(* Logix 5000 project; controller PBS_Perfusion vendor 1 type 14 code 217 rev 32.14; software revision 32.03; part 19 of 27 *)
(* tags used below, declared in another part *)
   Out_Open : BOOL;   // Pulse Output to drive valve Open
   Out_Close : BOOL;   // Pulse Output to drive valve closed
   P_ValveC : BOOL;   // Unique Parameter Name for auto - discovery
   OCmd_BumpClose : BOOL;   // Operator Command to bump valve closed (avail. if Fdbk Bad)
   OCmd_BumpOpen : BOOL;   // Operator Command to bump valve open (avail. if Fdbk Bad)
   ORdy_CV : BOOL;   // 1=Ready for OSet_CV (enables data entry field)
   ORdy_BumpClose : BOOL;   // 1=Ready for OCmd_BumpClose (enables HMI button)
   ORdy_BumpOpen : BOOL;   // 1=Ready for OCmd_BumpOpen (enables HMI button)
   REAL : DINT;
(* P_ValveC, continued *)

ROUTINE Prescan   (* ladder *)
// Clear Ownership. clear "lurking" Commands
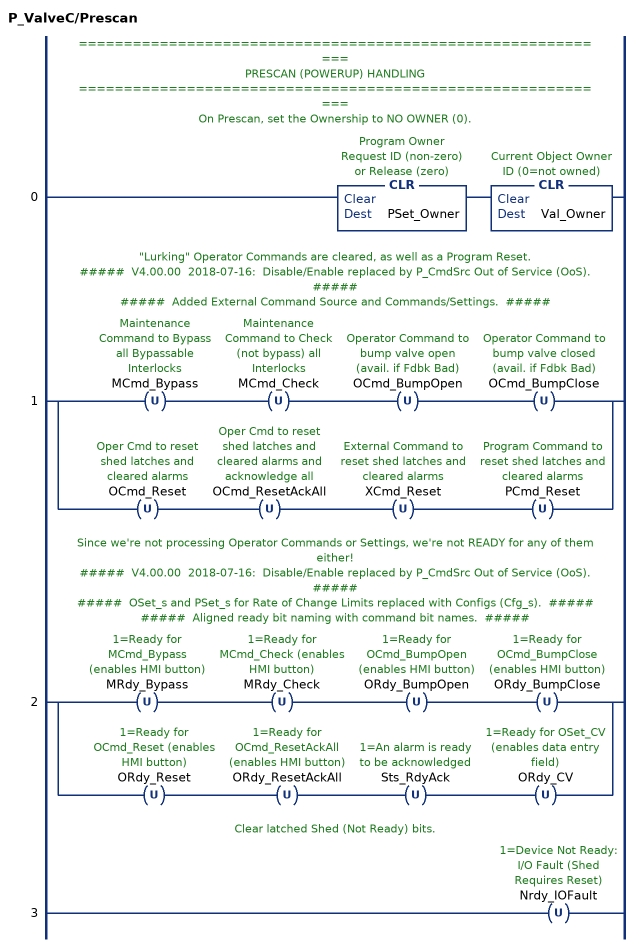
   // ============================================================
   // PRESCAN (POWERUP) HANDLING
   // ============================================================
   // On Prescan, set the Ownership to NO OWNER (0).
   0: CLR(PSet_Owner)CLR(Val_Owner);
   // "Lurking" Operator Commands are cleared, as well as a Program Reset.
   // #####  V4.00.00  2018-07-16:  Disable/Enable replaced by P_CmdSrc Out of Service (OoS).  #####
   // #####  Added External Command Source and Commands/Settings.  #####
   1: [OTU(MCmd_Bypass) OTU(MCmd_Check) OTU(OCmd_BumpOpen) OTU(OCmd_BumpClose) ,OTU(OCmd_Reset) OTU(OCmd_ResetAckAll) OTU(XCmd_Reset) OTU(PCmd_Reset) ];
   // Since we're not processing Operator Commands or Settings, we're not READY for any of them either!
   // #####  V4.00.00  2018-07-16:  Disable/Enable replaced by P_CmdSrc Out of Service (OoS).  #####
   // #####  OSet_s and PSet_s for Rate of Change Limits replaced with Configs (Cfg_s).  #####
   // #####  Aligned ready bit naming with command bit names.  #####
   2: [OTU(MRdy_Bypass) OTU(MRdy_Check) OTU(ORdy_BumpOpen) OTU(ORdy_BumpClose) ,OTU(ORdy_Reset) OTU(ORdy_ResetAckAll) OTU(Sts_RdyAck) OTU(ORdy_CV) ];
   // Clear latched Shed (Not Ready) bits.
   3: OTU(Nrdy_IOFault);
END_ROUTINE
END_ADD_ON_INSTRUCTION

ADD_ON_INSTRUCTION P_ValveSO   (* revision 4.10 .01 Release, vendor Rockwell Automation, ExecutePrescan, ExecuteEnableInFalse *)
// Solenoid Operated Valve
// Revision note:
// See Instruction Help for a summary of changes, and see 4.10 Release Notes for details.
// Help:
// Copyright © Rockwell Automation, Inc.  All Rights Reserved.
// This Instruction controls and monitors a single solenoid operated
// valve (two position: opened, closed) and provides:
// *  Support for fail open (energize to close) and fail closed (energize to open, default) valves
// *  Monitoring of limit switch feedback, display of actual valve status
// *  Detection of Failure to Open, Failure to Close
// *  Monitoring of Permissive conditions to allow energizing
// *  Monitoring of Interlock conditions to de-energize
// *  Simulation, providing feedback of a working valve while disabling outputs
// *  Monitoring of I/O communication faults
// *  Alarms for Full Stall (didn't move), Transit Stall (didn't reach target position), Interlock Trip, I/O Fault
// *  Operation in Hand, Maintenance, Override, Program and Operator Modes
// *  "Available" status for use by automation logic to know whether valve
//       can be controlled by other objects.
// Command Sources are arbitrated by a P_CmdSrc Add-On Instruction instance.
// Command Sources: Operator, External, Program, Override, Maintenance, Out of
// Service, Hand.  Alarms are provided by P_Alarm Add-On Instruction instances.
// SUMMARY OF CHANGES FROM PREVIOUS VERSION (4.10.00)
// See 4.10 Release Notes for details.
// * No changes, uprevved because P_CmdSrc 4.10.01 is used.
// SUMMARY OF CHANGES FROM PREVIOUS VERSION (4.00.02)
// See 4.10 Release Notes for details.
// * Added audible alert on commanded energize.
// * Added Horn Status, Horn Inhibit.
// * Updated to P_CmdSrc V4.10.00.
// * Added Cfg_HasMoreObj.
// SUMMARY OF CHANGES FROM PREVIOUS VERSION (4.00.01)
// See 4.00 Release Notes for details.
// * Modified handling of simultaneous open and close commands.
// SUMMARY OF CHANGES FROM PREVIOUS VERSION (4.00.00)
// See 4.00 Release Notes for details.
// * Corrected Reset Command logic.
// SUMMARY OF CHANGES FROM PREVIOUS VERSION (3.5-11)
// See 4.00 Release Notes for details.
// * Changed Inf_ items to HMI_, and added Cfg_Area for security.
// * Added notify and unack count rollup for Channel object.
// * Changed "Mode" to "Command Source" using P_CmdSrc 4.00.00.
// * Deleted Cfg_PCmdClear; all Program Commands are now self-clearing.
// * Aligned ready bit naming with command bit names.
// * All OCmds/MCmds and ORdys/MRdys are now Local Tags.
// * Added Sts_RdyAck and Sts_RdyReset for use by external objects.
// * Changed delay / time configuration items to REAL seconds.
VAR_INPUT
   Inp_OpenLS : BOOL; {visible}   // Valve Open Limit Switch 1=confirmed OPEN
   Inp_ClosedLS : BOOL; {visible}   // Valve Closed Limit Switch 1=confirmed CLOSED
   Inp_PermOK : BOOL := 1; {visible}   // 1=Permissives OK, Valve can energize
   Inp_NBPermOK : BOOL := 1; {visible}   // 1=Non-Bypassable Permissives OK, valve can energize
   Inp_IntlkOK : BOOL := 1; {visible}   // 1=Interlocks OK, valve can energize
   Inp_NBIntlkOK : BOOL := 1; {visible}   // 1=Non-Bypassable Interlocks OK, valve can energize
   Inp_IntlkAvail : BOOL;   // 1 = Interlock Availibility OK
   Inp_IOFault : BOOL;   // Input Communication Status 0=OK, 1=fail
   Inp_Sim : BOOL;   // 1=Simulate working valve; 0=Open/Close/ Monitor actual valve
   Inp_Hand : ALIAS FOR CmdSrc.Inp_Hand;
   Inp_Ovrd : ALIAS FOR CmdSrc.Inp_Ovrd;
   Inp_OvrdCmd : DINT;   // Override Mode Command: 0=None, 1=Close, 2=Open
   Inp_ExtInh : ALIAS FOR CmdSrc.Inp_ExtInh;
   Inp_HornInh : BOOL;   // 1 = Inhibit audible alert, 0 = Alllow audible alert
   Inp_Reset : BOOL;   // 1=Reset all fault conditions and latched Alarms
   Cfg_FailOpen : BOOL;   // 1=Fail Open (energize to close), 0=Fail Closed (energize to open)
   Cfg_HasOpenLS : BOOL;   // 1=Valve provides an Open Limit Switch signal
   Cfg_HasClosedLS : BOOL;   // 1=Valve provides a Closed Limit Switch signal
   Cfg_UseOpenLS : BOOL;   // 1=Valve Open LS should be used for failure checking
   Cfg_UseClosedLS : BOOL;   // 1=Valve Closed LS should be used for failure checking
   Cfg_LSFail : BOOL := 1;   // 1=both switches ON=fail, 0=both switches OFF=fail
   Cfg_HasPermObj : BOOL;   // 1=Tells HMI a P_Perm is connected to Inp_Perm
   Cfg_HasIntlkObj : BOOL;   // 1=Tells HMI a P_Intlk is connected to Inp_Intlk
   Cfg_HasStatsObj : BOOL;   // 1=Tells HMI a P_ValveStats is monitoring this valve
   Cfg_HasMoreObj : BOOL;   // 1=Tells HMI an object with more info is available
   Cfg_OCmdResets : BOOL;   // 1=New valve OCmd resets shed latches and cleared alarms, 0=OCmdReset req'd.
   Cfg_XCmdResets : BOOL;   // 1=New valve XCmd resets shed latches and cleared alarms, 0=OCmdReset req'd.
   Cfg_OvrdPermIntlk : BOOL;   // 1=Override ignores Bypassable Perm/ Intlk; 0=always use Perm/Intlk
   Cfg_ShedOnFullStall : BOOL := 1;   // 1=Stop Valve and Alarm on Full Stall; 0=Alarm only on Full Stall
   Cfg_ShedOnTransitStall : BOOL := 1;   // 1=Stop Valve and Alarm on Transit Stall; 0=Alarm only on Transit Stall
   Cfg_ShedOnIOFault : BOOL := 1;   // 1=Stop Valve and Alarm on I/O Fault; 0=Alarm only on I/O Fault
   Cfg_HasFullStallAlm : ALIAS FOR FullStall.Cfg_Exists;   // 1=Full Stall Alarm exists and will be checked
   Cfg_HasTransitStallAlm : ALIAS FOR TransitStall.Cfg_Exists;   // 1=Transit Stall Alarm exists and will be checked
   Cfg_HasIntlkTripAlm : ALIAS FOR IntlkTrip.Cfg_Exists;   // 1=Interlock Trip Alarm exists and will be checked
   Cfg_HasIOFaultAlm : ALIAS FOR IOFault.Cfg_Exists;   // 1=I/O Fault Alarm exists and will be checked
   Cfg_FullStallResetReqd : ALIAS FOR FullStall.Cfg_ResetReqd;   // 1=Reset requied to clear Full Stall Alarm
   Cfg_TransitStallResetReqd : ALIAS FOR TransitStall.Cfg_ResetReqd;   // 1=Reset required to clear Transit Stall Alarm
   Cfg_IntlkTripResetReqd : ALIAS FOR IntlkTrip.Cfg_ResetReqd;   // 1=Reset required to clear Interlock Trip Alarm
   Cfg_IOFaultResetReqd : ALIAS FOR IOFault.Cfg_ResetReqd;   // 1=Reset required to clear I/O Fault Alarm
   Cfg_FullStallAckReqd : ALIAS FOR FullStall.Cfg_AckReqd;   // 1=Acknowledge required for Full Stall Alarm
   Cfg_TransitStallAckReqd : ALIAS FOR TransitStall.Cfg_AckReqd;   // 1=Acknowledge required for Transit Stall Alarm
   Cfg_IntlkTripAckReqd : ALIAS FOR IntlkTrip.Cfg_AckReqd;   // 1=Acknowledge required for Interlock Trip Alarm
   Cfg_IOFaultAckReqd : ALIAS FOR IOFault.Cfg_AckReqd;   // 1=Acknowledge required for I/O Fault Alarm
   Cfg_FullStallSeverity : ALIAS FOR FullStall.Cfg_Severity;   // Full Stall Alarm Severity: 1..250=Low, 251..500=Medium, 501..750=High, 751..1000=Urgent
   Cfg_TransitStallSeverity : ALIAS FOR TransitStall.Cfg_Severity;   // Transit Stall Alarm Severity: 1..250=Low, 251..500=Medium, 501..750=High, 751..1000=Urgent
   Cfg_IntlkTripSeverity : ALIAS FOR IntlkTrip.Cfg_Severity;   // Interlock Trip Alarm Severity: 1..250=Low, 251..500=Medium, 501..750=High, 751..1000=Urgent
   Cfg_IOFaultSeverity : ALIAS FOR IOFault.Cfg_Severity;   // I/O Fault Alarm Severity: 1..250=Low, 251..500=Medium, 501..750=High, 751..1000=Urgent
   Cfg_SimFdbkT : REAL := 2.0;   // Delay to echo back of Open/Closed status when in Simulation (sec)
   Cfg_FullStallT : REAL := 5.0;   // After command, time with no motion before Fault (sec)
   Cfg_TransitStallT : REAL := 10.0;   // After command, time to reach position before fault (sec)
   Cfg_StartHornT : REAL;   // Time to sound audible on commanded start (sec) (0=disabled)
   PSet_Owner : DINT;   // Program Owner Request ID (non-zero) or Release (zero)
   PCmd_Open : BOOL;   // Program Command to Open Valve
   PCmd_Close : BOOL;   // Program Command to Close Valve
   PCmd_Prog : ALIAS FOR CmdSrc.PCmd_Prog;
   PCmd_Oper : ALIAS FOR CmdSrc.PCmd_Oper;
   PCmd_Lock : ALIAS FOR CmdSrc.PCmd_Lock;
   PCmd_Unlock : ALIAS FOR CmdSrc.PCmd_Unlock;
   PCmd_Normal : ALIAS FOR CmdSrc.PCmd_Normal;
   PCmd_Reset : BOOL;   // Program Command to ResetShed Latches and Cleared Alarms
   PCmd_FullStallAck : ALIAS FOR FullStall.PCmd_Ack;   // Program Command to Acknowledge Full Stall Alarm
   PCmd_FullStallSuppress : ALIAS FOR FullStall.PCmd_Suppress;   // Program Command to Suppress Full Stall Alarm
   PCmd_FullStallUnsuppress : ALIAS FOR FullStall.PCmd_Unsuppress;   // Program Command to Unsuppress Full Stall Alarm
   PCmd_FullStallUnshelve : ALIAS FOR FullStall.PCmd_Unshelve;   // Program Command to Unshelve Full Stall Alarm
   PCmd_TransitStallAck : ALIAS FOR TransitStall.PCmd_Ack;   // Program Command to Acknowledge Transit Stall Alarm
   PCmd_TransitStallSuppress : ALIAS FOR TransitStall.PCmd_Suppress;   // Program Command to Suppress Transit Stall Alarm
   PCmd_TransitStallUnsuppress : ALIAS FOR TransitStall.PCmd_Unsuppress;   // Program Command to Unsuppress Transit Stall Alarm
   PCmd_TransitStallUnshelve : ALIAS FOR TransitStall.PCmd_Unshelve;   // Program Command to Unshelve Transit Stall Alarm
   PCmd_IntlkTripAck : ALIAS FOR IntlkTrip.PCmd_Ack;   // Program Command to Acknowledge Interlock Trip Alarm
   PCmd_IntlkTripSuppress : ALIAS FOR IntlkTrip.PCmd_Suppress;   // Program Command to Suppress Interlock Trip Alarm
   PCmd_IntlkTripUnsuppress : ALIAS FOR IntlkTrip.PCmd_Unsuppress;   // Program Command to Unsuppress Interlock Trip Alarm
   PCmd_IntlkTripUnshelve : ALIAS FOR IntlkTrip.PCmd_Unshelve;   // Program Command to Unshelve Interlock Trip Alarm
   PCmd_IOFaultAck : ALIAS FOR IOFault.PCmd_Ack;   // Program Command to Acknowledge I/O Fault Alarm
   PCmd_IOFaultSuppress : ALIAS FOR IOFault.PCmd_Suppress;   // Program Command to Suppress I/O Fault Alarm
   PCmd_IOFaultUnsuppress : ALIAS FOR IOFault.PCmd_Unsuppress;   // Program Command to Unsuppress I/O Fault Alarm
   PCmd_IOFaultUnshelve : ALIAS FOR IOFault.PCmd_Unshelve;   // Program Command to Unshelve I/O Fault Alarm
   MCmd_Rel : ALIAS FOR CmdSrc.MCmd_Rel;
   OCmd_Unlock : ALIAS FOR CmdSrc.OCmd_Unlock;
   XCmd_Open : BOOL;   // External Command to Open Valve
   XCmd_Close : BOOL;   // External Command to Close Valve
   XCmd_Acq : ALIAS FOR CmdSrc.XCmd_Acq;
   XCmd_Rel : ALIAS FOR CmdSrc.XCmd_Rel;
   XCmd_Reset : BOOL;   // Ext Cmd to clear shed latches and cleared alarms
END_VAR
VAR_OUTPUT
   Out : BOOL; {access Read Only, visible}   // 1=Energize Valve Solenoid
   Out_Horn : BOOL; {access Read Only, visible}   // 1=Sound audible prior to commanded motor start
   SrcQ_IO : DINT; {access Read Only}   // Source and Quality of primary I/O (enumeration)
   SrcQ : DINT; {access Read Only}   // Source and Quality of primary Val/Sts (enumeration)
   Val_Cmd : DINT; {access Read Only}   // Device Command 0=None, 1=Close, 2=Open
   Val_Fdbk : DINT; {access Read Only}   // Device Feedback 0=Moving, 1=Closed, 2=Opened, 3=Limit Switch Failure
   Val_Sts : DINT; {access Read Only}   // Device Confirmed Sts 0=? 1=Closed 2=Open 5=Closing, 6=Opening
   Val_Fault : DINT; {access Read Only}   // Device Fault Status 0=None, 16=Transit Stall, 17 = Full Stall, 32=I/O Fault, 34=Config Error
   Val_NotifyAll : DINT; {access Read Only}   // Highest Alarm prio and ack status this object + channel (enum)
   Val_UnackAlmC : DINT; {access Read Only}   // Count of Unacknowledged Alarms
   Val_Owner : DINT; {access Read Only}   // Current Object Owner ID (0=not owned)
   Sts_Closed : BOOL; {access Read Only, visible}   // 1=Valve requested to Close and is confirmed Closed
   Sts_Opening : BOOL; {access Read Only, visible}   // 1=Valve requested to open and awaiting open feedback
   Sts_Opened : BOOL; {access Read Only, visible}   // 1=Valve requested to open and is confirmed Opened
   Sts_Closing : BOOL; {access Read Only, visible}   // 1=Valve requested to Close and awaiting Closed feedback
   Sts_Horn : BOOL; {access Read Only}   // 1=Valve Horn Active
   Sts_Available : BOOL; {access Read Only}   // 1=Valve available for control by automation (Prog)
   Sts_Bypass : BOOL; {access Read Only}   // 1=Bypassable Interlocks and Permissives are Bypassed
   Sts_BypActive : BOOL; {access Read Only}   // 1=Bypassing Active (Bypassed or Maintenance)
   Sts_LSFail : BOOL; {access Read Only}   // 1=Limit Switch Overlap Failure
   Sts_NotRdy : BOOL; {access Read Only}   // 1=Device Not Ready, see detail bits for reason
   Nrdy_CfgErr : BOOL; {access Read Only}   // 1=Device Not Ready: Configuration Error
   Nrdy_Fail : BOOL; {access Read Only}   // 1=Device Not Ready: Device Failure (Shed Requires Reset)
   Nrdy_Intlk : BOOL; {access Read Only}   // 1=Device Not Ready: Interlock Not OK
   Nrdy_IOFault : BOOL; {access Read Only}   // 1=Device Not Ready: I/O Fault (Shed Requires Reset)
   Nrdy_OoS : BOOL; {access Read Only}   // 1=Device Not Ready: Device is Out of Service
   Nrdy_Perm : BOOL; {access Read Only}   // 1=Device Not Ready: Permissive Not OK
   Sts_MaintByp : BOOL; {access Read Only}   // 1=A Maintenance Bypass is Active, display icon
   Sts_AlmInh : BOOL; {access Read Only}   // 1=An Alarm is Shelved, Disabled or Suppressed, display icon
   Sts_Err : BOOL; {access Read Only, visible}   // 1=Error in Config: see detail bits for reason
   Err_Timer : BOOL; {access Read Only}   // 1=Error in Config: Invalid Check Time (use 0 to 2147483)
   Err_Sim : BOOL; {access Read Only}   // 1=Error in Config: Invalid Simulation Time (use 0 to 2147483)
   Err_Alarm : BOOL; {access Read Only}   // 1=Error in Config: Alarm Min On Time, Shelf Time, Severity
   Sts_Hand : ALIAS FOR CmdSrc.Sts_Hand; {access Read Only, visible}
   Sts_OoS : ALIAS FOR CmdSrc.Sts_OoS; {access Read Only, visible}
   Sts_Maint : ALIAS FOR CmdSrc.Sts_Maint; {access Read Only, visible}
   Sts_Ovrd : ALIAS FOR CmdSrc.Sts_Ovrd; {access Read Only, visible}
   Sts_Ext : ALIAS FOR CmdSrc.Sts_Ext; {access Read Only, visible}
   Sts_Prog : ALIAS FOR CmdSrc.Sts_Prog; {access Read Only, visible}
   Sts_ProgLocked : ALIAS FOR CmdSrc.Sts_ProgLocked; {access Read Only}
   Sts_Oper : ALIAS FOR CmdSrc.Sts_Oper; {access Read Only, visible}
   Sts_OperLocked : ALIAS FOR CmdSrc.Sts_OperLocked; {access Read Only}
   Sts_Normal : ALIAS FOR CmdSrc.Sts_Normal; {access Read Only}
   Sts_ExtReqInh : ALIAS FOR CmdSrc.Sts_ExtReqInh; {access Read Only}
   Sts_ProgReqInh : ALIAS FOR CmdSrc.Sts_ProgReqInh; {access Read Only}
   Sts_MAcqRcvd : ALIAS FOR CmdSrc.Sts_MAcqRcvd; {access Read Only}
   Sts_RdyReset : ALIAS FOR ORdy_Reset; {access Read Only}   // 1=A latched alarm or shed condition is ready to be reset
   Sts_RdyAck : BOOL; {access Read Only}   // 1=An alarm is ready to be acknowledged
   Sts_FullStall : ALIAS FOR FullStall.Inp;   // 1=Valve Full Stall (failed to move at all)
   Alm_FullStall : ALIAS FOR FullStall.Alm;   // 1=Valve Full Stall (failed to move at all) Alarm
   Ack_FullStall : ALIAS FOR FullStall.Ack;   // 1=Full Stall Alarm has been acknowledged
   Sts_FullStallDisabled : ALIAS FOR FullStall.Disabled;   // 1=Full Stall Alarm has been Disabled by Maintenance
   Sts_FullStallShelved : ALIAS FOR FullStall.Shelved;   // 1=Full Stall Alarm has been Shelved by Operator
   Sts_FullStallSuppressed : ALIAS FOR FullStall.Suppressed;   // 1=Full Stall Alarm has been Suppressed by Program
   Sts_TransitStall : ALIAS FOR TransitStall.Inp;   // 1=Valve Transit Stall (did not reach target position)
   Alm_TransitStall : ALIAS FOR TransitStall.Alm;   // 1=Valve Transit Stall (did not reach target pos.) Alarm
   Ack_TransitStall : ALIAS FOR TransitStall.Ack;   // 1=Transit Stall Alarm has been acknowledged
   Sts_TransitStallDisabled : ALIAS FOR TransitStall.Disabled;   // 1=Transit Stall Alarm has been Disabled by Maintenance
   Sts_TransitStallShelved : ALIAS FOR TransitStall.Shelved;   // 1=Transit Stall Alarm has been Shelved by Operator
   Sts_TransitStallSuppressed : ALIAS FOR TransitStall.Suppressed;   // 1=Transit Stall Alarm has been Suppressed by Program
   Sts_IntlkTrip : ALIAS FOR IntlkTrip.Inp;   // 1=Valve de-energized by an Interlock NOT OK
   Alm_IntlkTrip : ALIAS FOR IntlkTrip.Alm;   // 1=Alarm: Valve de-energized by an Interlock NOT OK
   Ack_IntlkTrip : ALIAS FOR IntlkTrip.Ack;   // 1=Interlock Trip Alarm has been acknowledged
   Sts_IntlkTripDisabled : ALIAS FOR IntlkTrip.Disabled;   // 1=Interlock Trip Alarm has been Disabled by Maintenance
   Sts_IntlkTripShelved : ALIAS FOR IntlkTrip.Shelved;   // 1=Interlock Trip Alarm has been Shelved by Operator
   Sts_IntlkTripSuppressed : ALIAS FOR IntlkTrip.Suppressed;   // 1=Interlock Trip Alarm has been Suppressed Program
   Sts_IOFault : ALIAS FOR IOFault.Inp;   // I/O Comm Fault Status (0=OK, 1=Bad)
   Alm_IOFault : ALIAS FOR IOFault.Alm;   // 1=I/O Fault Alarm
   Ack_IOFault : ALIAS FOR IOFault.Ack;   // 1=I/O Fault Alarm has been acknowledged
   Sts_IOFaultDisabled : ALIAS FOR IOFault.Disabled;   // 1=I/O Fault Alarm has been Disabled by Maintenance
   Sts_IOFaultShelved : ALIAS FOR IOFault.Shelved;   // 1=I/O Fault Alarm has been Shelved by Operator
   Sts_IOFaultSuppressed : ALIAS FOR IOFault.Suppressed;   // 1=I/O Fault Alarm has been Suppressed by Program
   MRdy_Rel : ALIAS FOR CmdSrc.MRdy_Rel; {access Read Only}
   ORdy_Unlock : ALIAS FOR CmdSrc.ORdy_Unlock; {access Read Only}
   P_ValveSO : BOOL;   // Unique Parameter Name for auto - discovery
END_VAR
VAR
   CmdSrc : P_CmdSrc := (Cfg_HasOper := 1, Cfg_HasOperLocked := 1, Cfg_HasProg := 1, Cfg_HasProgLocked := 1, Cfg_HasMaint := 1, Cfg_HasMOoS := 1, Cfg_OvrdOverLock := 1, Sts_bSrc := 1);   // Valve Mode Selection
   IOFault : P_Alarm := (Cfg_AckReqd := 1, Cfg_AllowShelve := 1, Cfg_AllowDisable := 1, Cfg_Severity := 1000, Cfg_AlmMinOnT := 5, PCfg_AllowExist := 1, Ack := 1);   // I/O Fault Alarm
   IntlkTrip : P_Alarm := (Cfg_AckReqd := 1, Cfg_AllowShelve := 1, Cfg_AllowDisable := 1, Cfg_Severity := 500, Cfg_AlmMinOnT := 5, PCfg_AllowExist := 1, Ack := 1);   // Interlock Trip Alarm
   TransitStall : P_Alarm := (Cfg_AckReqd := 1, Cfg_AllowShelve := 1, Cfg_AllowDisable := 1, Cfg_Severity := 1000, Cfg_AlmMinOnT := 5, PCfg_AllowExist := 1, Ack := 1);   // Valve Transit Stall (moved but did not reach target) Alarm
   FullStall : P_Alarm := (Cfg_AckReqd := 1, Cfg_AllowShelve := 1, Cfg_AllowDisable := 1, Cfg_Severity := 1000, Cfg_AlmMinOnT := 5, PCfg_AllowExist := 1, Ack := 1);   // Valve Full Stall (did not move) Alarm
   Cfg_Tag : STRING_20 := 'P_ValveSO';   // Tagname for display on HMI
   Cfg_Label : STRING_20 := 'Valve Control';   // Label for graphic symbol displayed on HMI
   Cfg_Desc : STRING_40 := 'Solenoid Operated Valve';   // Description for display on HMI
   Wrk_Open : BOOL; {access None}   // 1=Requested to OPEN Valve, 0=Requested to CLOSE Valve
   Wrk_SimOpenT : TIMER; {access None}   // Simulation Delay until Opened
   Wrk_SimCloseT : TIMER; {access None}   // Simulation Delay until Closed
   Wrk_OpenFdbk : BOOL; {access None}   // 1=LS Feedback shows valve confirmed open
   Wrk_Notify : DINT; {access None}   // Buffer for building Val_Notify
   Wrk_Bypass : BOOL; {access None}   // Internal Bypassable Permissives and Interlocks are Bypassed flag
   Wrk_ClosedFdbk : BOOL; {access None}   // 1=LS Feedback shows valve confirmed closed
   Wrk_TransitStallT : TIMER; {access Read Only}   // Timer for Transit Stall Check
   Wrk_FullStallT : TIMER; {access Read Only}   // Timer for Full Stall Check
   HMI_Tab : SINT;   // Tab to display (FTView ME)
   Wrk_Cmd : DINT; {access None}   // Buffer for building Val_Cmd
   Wrk_Sts : DINT; {access None}   // Buffer for building Val_Sts
   Wrk_Fault : DINT; {access None}   // Buffer for building Val_Fault
   HMI_Type : STRING_16 := 'P_ValveSO'; {access Read Only}   // Type identifier for HMI navigation
   Wrk_SimOpenLS : BOOL; {access None}   // Simulated valve Open Limit Switch
   Wrk_SimClosedLS : BOOL; {access None}   // Simulated valve Closed Limit Switch
   HMI_Lib : STRING_12 := 'RA-BAS'; {access Read Only}   // Display Library for Faceplate call-up
   Wrk_SrcQ : DINT; {access None}   // Register for building Source / Quality enumeration
   Val_Notify : DINT; {access Read Only}   // Current Alarm Level and Acknowledgement (enumeration)
   Wrk_NotRdy : BOOL; {access None}   // Device Not Ready conditions excluding shed latches
   Wrk_NoLongerSim : BOOL; {access None}   // Switched from Simulated to Real Valve this scan
   OCmd_Close : BOOL;   // Operator Command to Close Valve
   OCmd_Open : BOOL;   // Operator Command to Open Valve
   ORdy_ResetAckAll : BOOL; {access Read Only}   // 1=Ready for OCmd_ResetAckAll (enables HMI button)
   ORdy_Reset : BOOL; {access Read Only}   // 1=Ready for OCmd_Reset (enables HMI button)
   MRdy_Check : BOOL; {access Read Only}   // 1=Ready for MCmd_Check (enables HMI button)
   MRdy_Bypass : BOOL; {access Read Only}   // 1=Ready for MCmd_Bypass (enables HMI button)
   ORdy_Close : BOOL; {access Read Only}   // 1=Ready for OCmd_Close (enables HMI button)
   ORdy_Open : BOOL; {access Read Only}   // 1=Ready for OCmd_Open (enables HMI button)
   MCmd_Check : BOOL;   // Maintenance Command to Check (not bypass) all Interlocks and Permissives
   MCmd_Bypass : BOOL;   // Maintenance Command to Bypass all Bypassable Interlocks and Permissives
   Cfg_Area : STRING_Area := 'area01';   // Process Area for security
   OCmd_ResetAckAll : BOOL;   // Oper Cmd to reset shed latches and cleared alarms, plus Acknowledge alarms
   OCmd_Reset : BOOL;   // Oper Cmd to clear shed latches and cleared alarms
   Wrk_UnackAlmC : DINT; {access None}   // Buffer for building Val_UnackAlmC
   Wrk_CloseCmdRcvd : BOOL; {access None}   // 1=Received a Close command this scan
   Wrk_OpenCmdRcvd : BOOL; {access None}   // 1=Received an Open command this scan
   Wrk_StartHornT : TIMER; {access None}   // Timer for audible alert on start
   Wrk_StartHorn : BOOL; {access None}   // 1=Sound audible prior to commanded motor start
END_VAR

ROUTINE EnableInFalse   (* ladder *)
// Out of Service is asserted; Outputs OFF; Valve Status shown but Alarms inhibited.
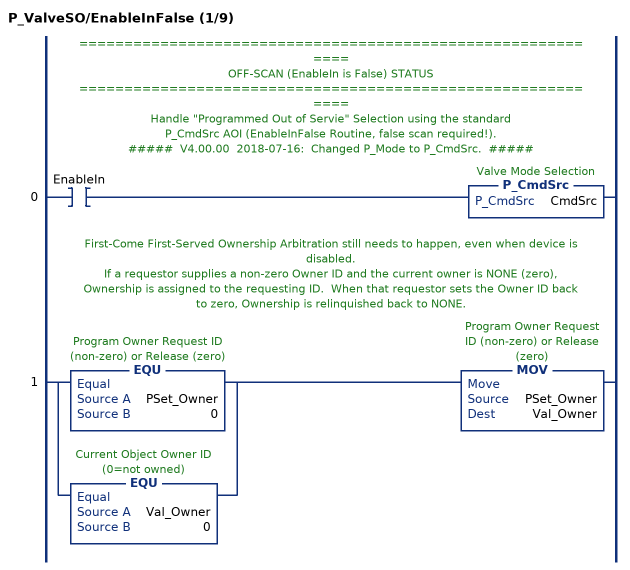
   // ============================================================
   // OFF-SCAN (EnableIn is False) STATUS
   // ============================================================
   // Handle "Programmed Out of Servie" Selection using the standard
   // P_CmdSrc AOI (EnableInFalse Routine, false scan required!).
   // #####  V4.00.00  2018-07-16:  Changed P_Mode to P_CmdSrc.  #####
   0: XIC(EnableIn)P_CmdSrc(CmdSrc);
   // First-Come First-Served Ownership Arbitration still needs to happen, even when device is disabled.
   // If a requestor supplies a non-zero Owner ID and the current owner is NONE (zero),
   // Ownership is assigned to the requesting ID.  When that requestor sets the Owner ID back
   // to zero, Ownership is relinquished back to NONE.
   1: [EQU(PSet_Owner,0) ,EQU(Val_Owner,0) ]MOV(PSet_Owner,Val_Owner);
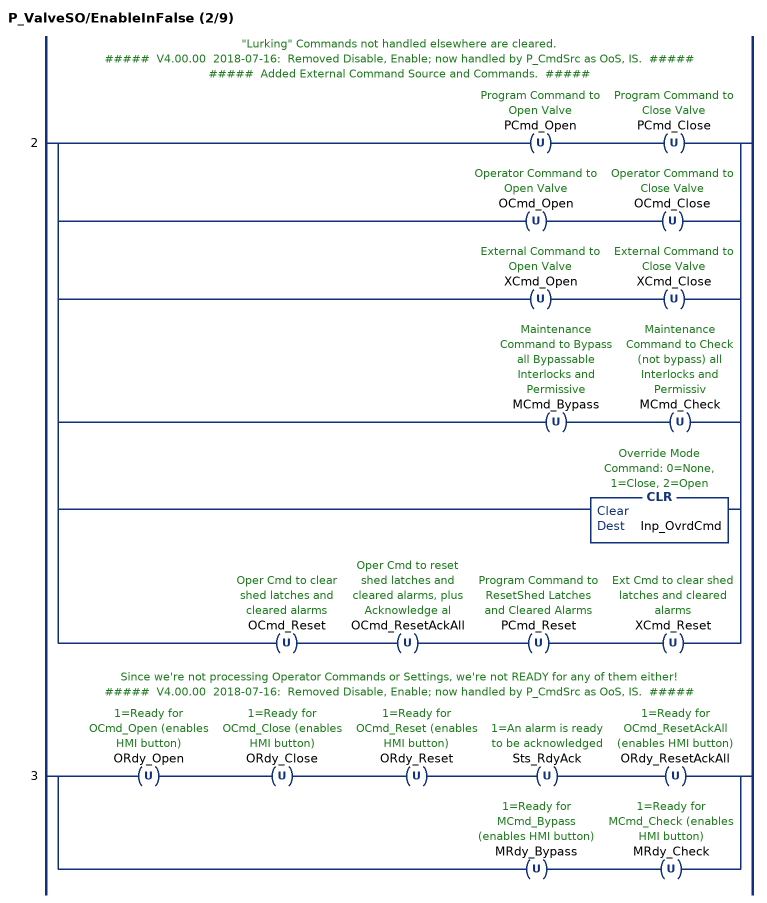
   // "Lurking" Commands not handled elsewhere are cleared.
   // #####  V4.00.00  2018-07-16:  Removed Disable, Enable; now handled by P_CmdSrc as OoS, IS.  #####
   // #####  Added External Command Source and Commands.  #####
   2: [OTU(PCmd_Open) OTU(PCmd_Close) ,OTU(OCmd_Open) OTU(OCmd_Close) ,OTU(XCmd_Open) OTU(XCmd_Close) ,OTU(MCmd_Bypass) OTU(MCmd_Check) ,CLR(Inp_OvrdCmd) ,OTU(OCmd_Reset) OTU(OCmd_ResetAckAll) OTU(PCmd_Reset) OTU(XCmd_Reset) ];
   // Since we're not processing Operator Commands or Settings, we're not READY for any of them either!
   // #####  V4.00.00  2018-07-16:  Removed Disable, Enable; now handled by P_CmdSrc as OoS, IS.  #####
   3: [OTU(ORdy_Open) OTU(ORdy_Close) OTU(ORdy_Reset) OTU(Sts_RdyAck) OTU(ORdy_ResetAckAll) ,OTU(MRdy_Bypass) OTU(MRdy_Check) ];
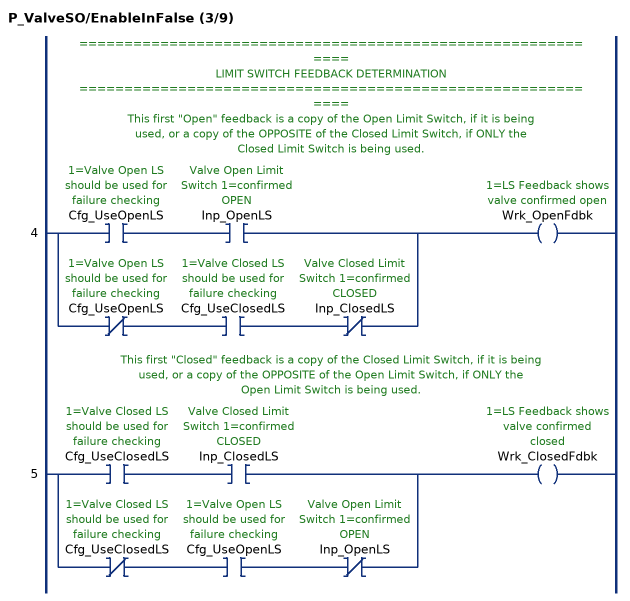
   // ============================================================
   // LIMIT SWITCH FEEDBACK DETERMINATION
   // ============================================================
   // This first "Open" feedback is a copy of the Open Limit Switch, if it is being
   // used, or a copy of the OPPOSITE of the Closed Limit Switch, if ONLY the
   // Closed Limit Switch is being used.
   4: [XIC(Cfg_UseOpenLS) XIC(Inp_OpenLS) ,XIO(Cfg_UseOpenLS) XIC(Cfg_UseClosedLS) XIO(Inp_ClosedLS) ]OTE(Wrk_OpenFdbk);
   // This first "Closed" feedback is a copy of the Closed Limit Switch, if it is being
   // used, or a copy of the OPPOSITE of the Open Limit Switch, if ONLY the
   // Open Limit Switch is being used.
   5: [XIC(Cfg_UseClosedLS) XIC(Inp_ClosedLS) ,XIO(Cfg_UseClosedLS) XIC(Cfg_UseOpenLS) XIO(Inp_OpenLS) ]OTE(Wrk_ClosedFdbk);
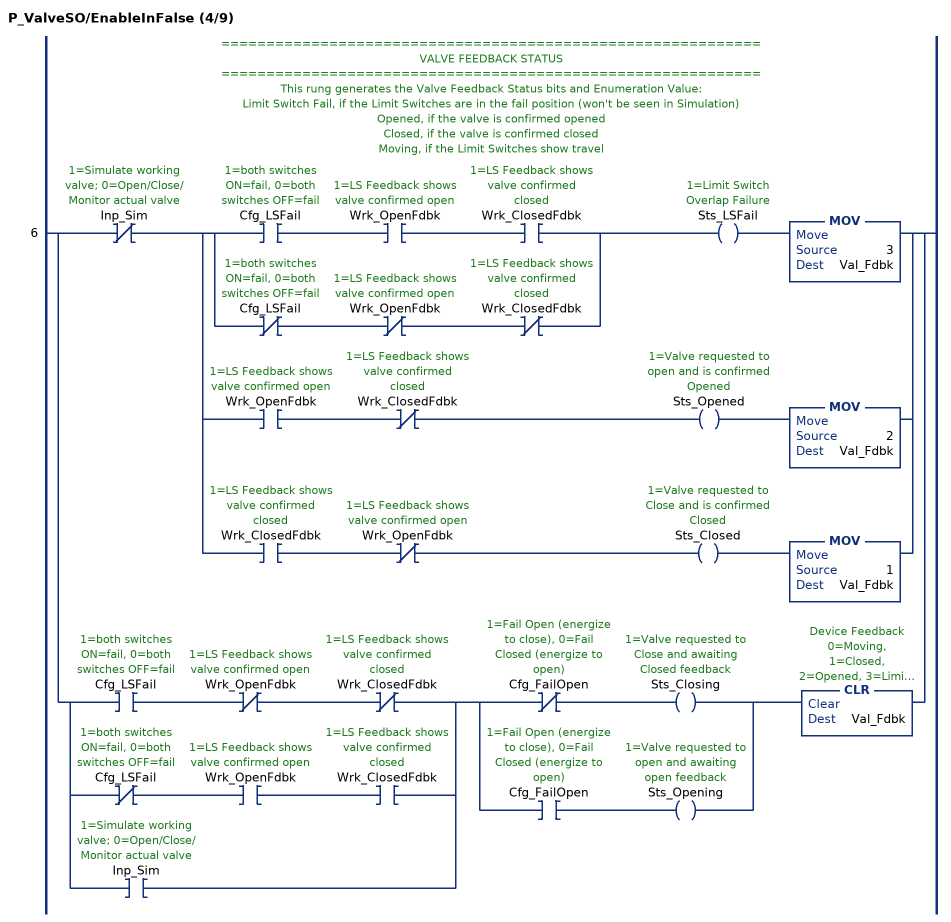
   // ============================================================
   // VALVE FEEDBACK STATUS
   // ============================================================
   // This rung generates the Valve Feedback Status bits and Enumeration Value:
   // Limit Switch Fail, if the Limit Switches are in the fail position (won't be seen in Simulation)
   // Opened, if the valve is confirmed opened
   // Closed, if the valve is confirmed closed
   // Moving, if the Limit Switches show travel
   6: [XIO(Inp_Sim) [[XIC(Cfg_LSFail) XIC(Wrk_OpenFdbk) XIC(Wrk_ClosedFdbk) ,XIO(Cfg_LSFail) XIO(Wrk_OpenFdbk) XIO(Wrk_ClosedFdbk) ] OTE(Sts_LSFail) MOV(3,Val_Fdbk) ,XIC(Wrk_OpenFdbk) XIO(Wrk_ClosedFdbk) OTE(Sts_Opened) MOV(2,Val_Fdbk) ,XIC(Wrk_ClosedFdbk) XIO(Wrk_OpenFdbk) OTE(Sts_Closed) MOV(1,Val_Fdbk) ] ,[[XIC(Cfg_LSFail) XIO(Wrk_OpenFdbk) XIO(Wrk_ClosedFdbk) ,XIO(Cfg_LSFail) XIC(Wrk_OpenFdbk) XIC(Wrk_ClosedFdbk) ] ,XIC(Inp_Sim) ] [XIO(Cfg_FailOpen) OTE(Sts_Closing) ,XIC(Cfg_FailOpen) OTE(Sts_Opening) ] CLR(Val_Fdbk) ];
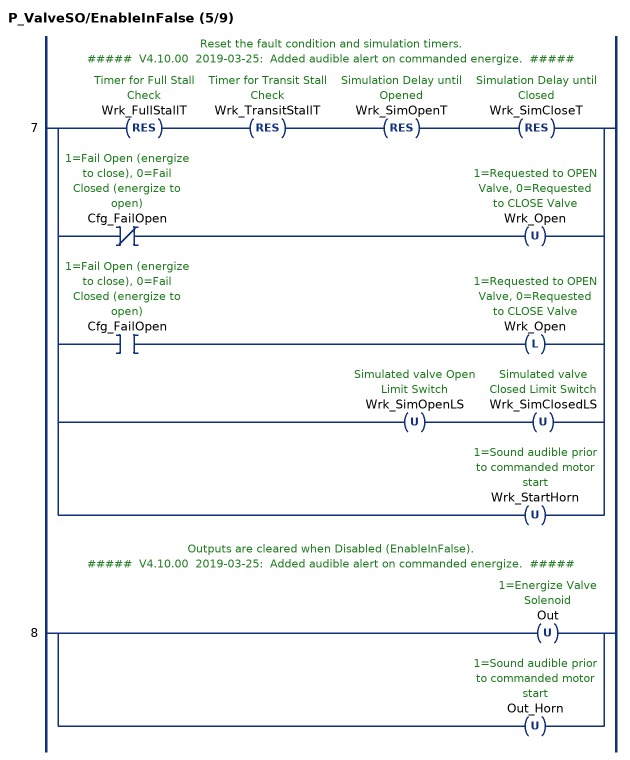
   // Reset the fault condition and simulation timers.
   // #####  V4.10.00  2019-03-25:  Added audible alert on commanded energize.  #####
   7: [RES(Wrk_FullStallT) RES(Wrk_TransitStallT) RES(Wrk_SimOpenT) RES(Wrk_SimCloseT) ,[XIO(Cfg_FailOpen) OTU(Wrk_Open) ,XIC(Cfg_FailOpen) OTL(Wrk_Open) ] ,OTU(Wrk_SimOpenLS) OTU(Wrk_SimClosedLS) ,OTU(Wrk_StartHorn) ];
   // Outputs are cleared when Disabled (EnableInFalse).
   // #####  V4.10.00  2019-03-25:  Added audible alert on commanded energize.  #####
   8: [OTU(Out) ,OTU(Out_Horn) ];
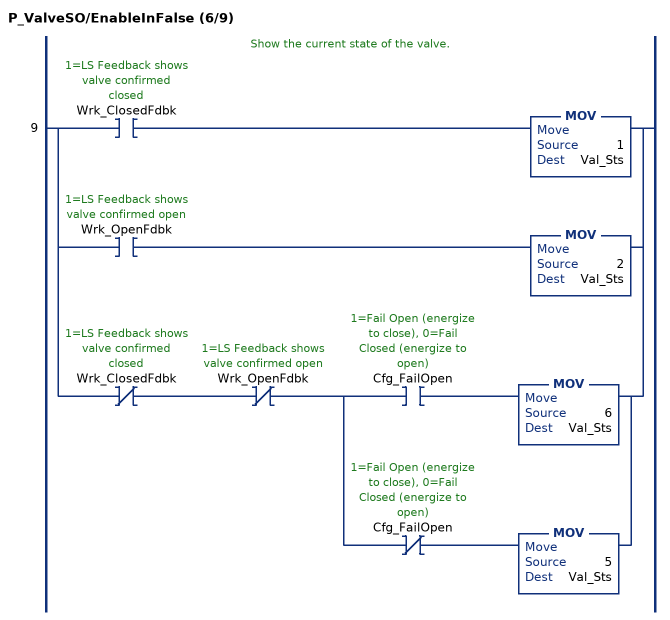
   // Show the current state of the valve.
   9: [XIC(Wrk_ClosedFdbk) MOV(1,Val_Sts) ,XIC(Wrk_OpenFdbk) MOV(2,Val_Sts) ,XIO(Wrk_ClosedFdbk) XIO(Wrk_OpenFdbk) [XIC(Cfg_FailOpen) MOV(6,Val_Sts) ,XIO(Cfg_FailOpen) MOV(5,Val_Sts) ] ];
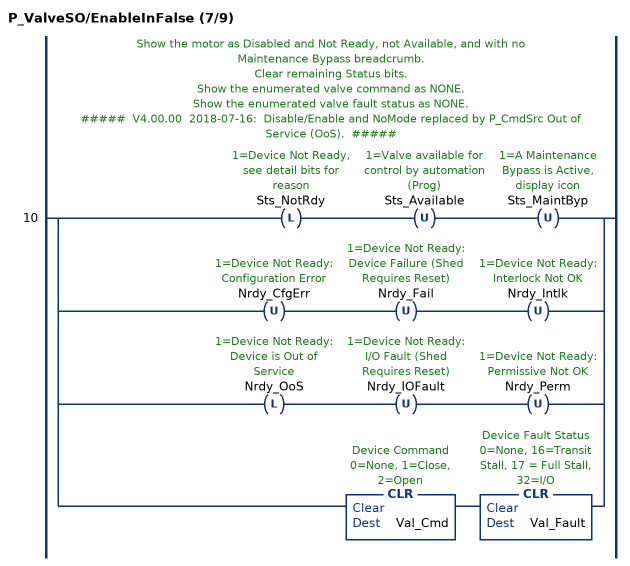
   // Show the motor as Disabled and Not Ready, not Available, and with no
   // Maintenance Bypass breadcrumb.
   // Clear remaining Status bits.
   // Show the enumerated valve command as NONE.
   // Show the enumerated valve fault status as NONE.
   // #####  V4.00.00  2018-07-16:  Disable/Enable and NoMode replaced by P_CmdSrc Out of Service (OoS).  #####
   10: [OTL(Sts_NotRdy) OTU(Sts_Available) OTU(Sts_MaintByp) ,OTU(Nrdy_CfgErr) OTU(Nrdy_Fail) OTU(Nrdy_Intlk) ,OTL(Nrdy_OoS) OTU(Nrdy_IOFault) OTU(Nrdy_Perm) ,CLR(Val_Cmd) CLR(Val_Fault) ];
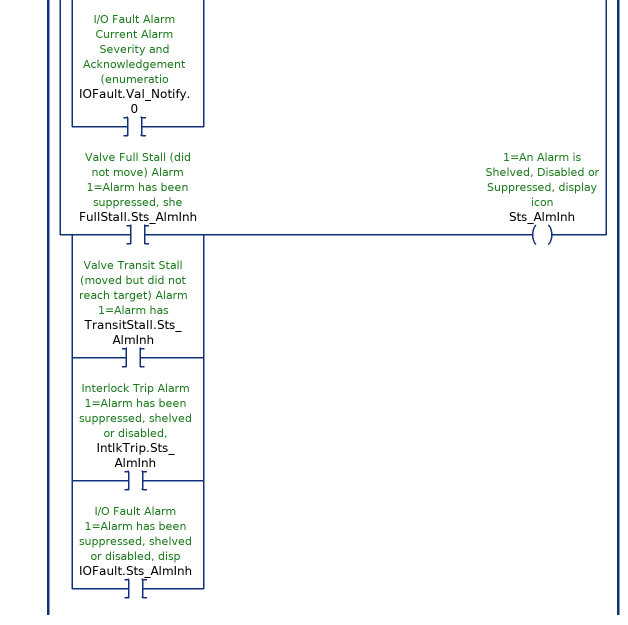
   // If this Analog Output is OFF-SCAN (rung is false or EnableIn is false in FBD),
   // then show the alarms as "Parent object out of service".
   // Show the overall acknowledgement status.
   // #####  V4.00.00  2018-07-16:  Changed P_Mode to P_CmdSrc, added Out of Service.  #####
   11: [OTL(FullStall.Inp_OoS) P_Alarm(FullStall) ,OTL(TransitStall.Inp_OoS) P_Alarm(TransitStall) ,OTL(IntlkTrip.Inp_OoS) P_Alarm(IntlkTrip) ,OTL(IOFault.Inp_OoS) P_Alarm(IOFault) ,CLR(Val_Notify) CLR(Val_NotifyAll) ,[XIC(FullStall.Val_Notify.0) ,XIC(TransitStall.Val_Notify.0) ,XIC(IntlkTrip.Val_Notify.0) ,XIC(IOFault.Val_Notify.0) ] OTL(Val_Notify.0) OTL(Val_NotifyAll.0) ,[XIC(FullStall.Sts_AlmInh) ,XIC(TransitStall.Sts_AlmInh) ,XIC(IntlkTrip.Sts_AlmInh) ,XIC(IOFault.Sts_AlmInh) ] OTE(Sts_AlmInh) ];
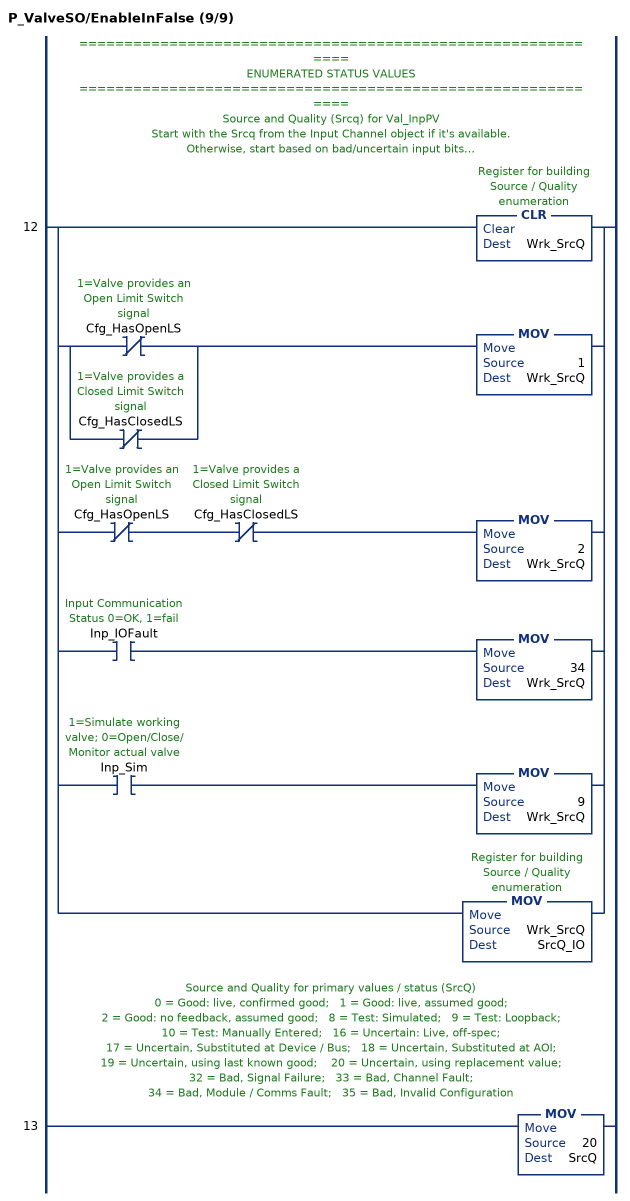
   // ============================================================
   // ENUMERATED STATUS VALUES
   // ============================================================
   // Source and Quality (Srcq) for Val_InpPV
   // Start with the Srcq from the Input Channel object if it's available.
   // Otherwise, start based on bad/uncertain input bits.
   // 0 = Good: live, confirmed good;   1 = Good: live, assumed good;
   // 2 = Good: no feedback, assumed good;   8 = Test: Simulated;   9 = Test: Loopback;
   // 10 = Test: Manually Entered;   16 = Uncertain: Live, off-spec;
   // 17 = Uncertain, Substituted at Device / Bus;   18 = Uncertain, Substituted at AOI;
   // 19 = Uncertain, using last known good;    20 = Uncertain, using replacement value;
   // 32 = Bad, Signal Failure;   33 = Bad, Channel Fault;
   // 34 = Bad, Module / Comms Fault;   35 = Bad, Invalid Configuration
   12: [CLR(Wrk_SrcQ) ,[XIO(Cfg_HasOpenLS) ,XIO(Cfg_HasClosedLS) ] MOV(1,Wrk_SrcQ) ,XIO(Cfg_HasOpenLS) XIO(Cfg_HasClosedLS) MOV(2,Wrk_SrcQ) ,XIC(Inp_IOFault) MOV(34,Wrk_SrcQ) ,XIC(Inp_Sim) MOV(9,Wrk_SrcQ) ,MOV(Wrk_SrcQ,SrcQ_IO) ];
   // Source and Quality for primary values / status (SrcQ)
   // 0 = Good: live, confirmed good;   1 = Good: live, assumed good;
   // 2 = Good: no feedback, assumed good;   8 = Test: Simulated;   9 = Test: Loopback;
   // 10 = Test: Manually Entered;   16 = Uncertain: Live, off-spec;
   // 17 = Uncertain, Substituted at Device / Bus;   18 = Uncertain, Substituted at AOI;
   // 19 = Uncertain, using last known good;    20 = Uncertain, using replacement value;
   // 32 = Bad, Signal Failure;   33 = Bad, Channel Fault;
   // 34 = Bad, Module / Comms Fault;   35 = Bad, Invalid Configuration
   13: MOV(20,SrcQ);
END_ROUTINE

ROUTINE Logic   (* ladder *)
// Normal Scan: control / monitor solenoid-operated valve
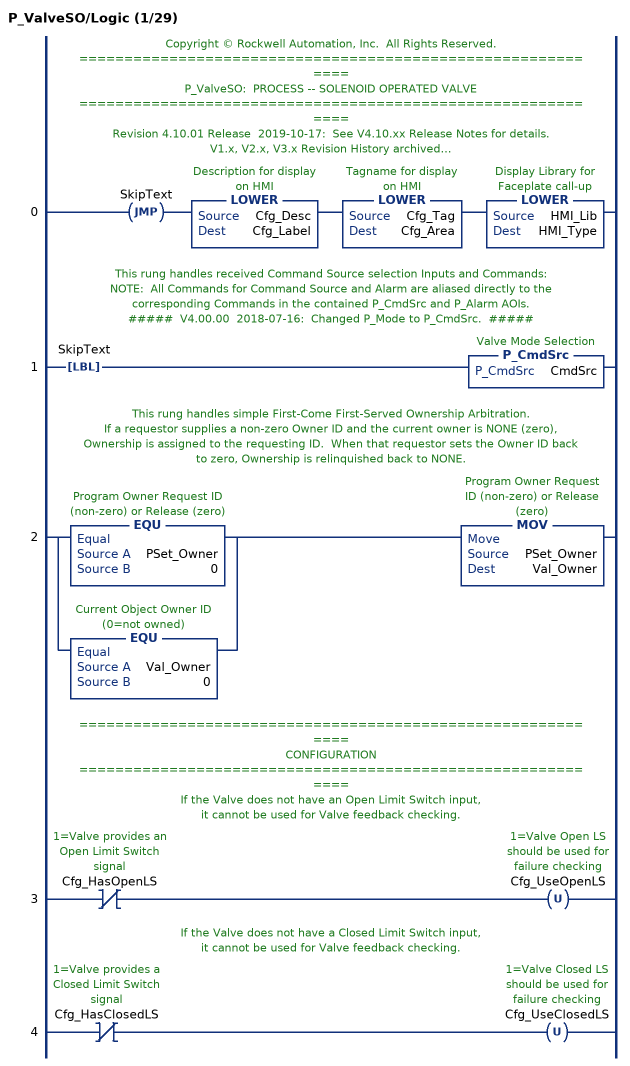
   // Copyright © Rockwell Automation, Inc.  All Rights Reserved.
   // ============================================================
   // P_ValveSO:  PROCESS -- SOLENOID OPERATED VALVE
   // ============================================================
   // Revision 4.10.01 Release  2019-10-17:  See V4.10.xx Release Notes for details.
   // V1.x, V2.x, V3.x Revision History archived.
   // V4.00.00  2018-07-16:  Changed "Mode" to "Command Source". Changed Inf_ items
   // to HMI_, and added Cfg_Area for security. Added unacked alarm count.
   // Deleted Cfg_PCmdClear; all Program Commands are now self-clearing.
   // Aligned ready bit naming with command bit names.
   // Changed delay / time configuration items to REAL seconds.
   // V4.00.01  2018-08-24:  Corrected Reset Command logic.
   // V4.00.02  2018-11-02:  Modified handling of simultaneous open and close commands.
   // V4.10.00  2019-03-25:  Added audible alert on commanded energize. Added Horn
   // Status, Horn Inhibit. Updated to P_CmdSrc V4.10.00. Added Cfg_HasMoreObj.
   // V4.10.01  2019-10-17:  No changes, uprevved because P_CmdSrc 4.10.01 is used.
   // ============================================================
   // This Instruction controls and monitors a single solenoid operated
   // valve (typ. two position: opened, closed) and provides:
   // *  Support for fail open (energize to close) and fail closed (energize to open, default) valves
   // *  Monitoring of limit switch feedback, display of actual valve status
   // *  Detection of failure to move (full stall), failure to reach position (transit stall)
   // *  Monitoring of Permissive conditions to allow energizing
   // *  Monitoring of Interlock conditions to de-energize
   // *  Simulation, providing feedback of a working valve while disabling outputs
   // *  Monitoring of I/O communication faults
   // *  Alarms for Full Stall, Transit Stall, Interlock Trip, I/O Fault
   // *  "Available" status for use by automation logic to know whether valve
   // can be controlled by other objects.
   // Command Sources are arbitrated by a P_CmdSrc Add-On Instruction instance.
   // Command Sources: Operator, External, Program, External, Override, Maintenance,
   // Out of Service, Hand.  Alarms are provided by P_Alarm Add-On Instruction instances.
   // ============================================================
   // SHOW LOCAL STRINGS
   // ============================================================
   // The STRINGs containing the text associated with each instance of this
   // instruction cannot be Input or Output Parameters, because STRINGs are not
   //  'atomic' types. (Inputs and Outputs must be SINT, INT, DINT, REAL, or BOOL.)
   // In order to make it easier to find and configure these STRINGs, this rung
   // was added.  THE JMP (and the LBL on the following rung)
   // MUST NOT BE REMOVED!!!
   // To view the STRINGs, go to the instruction instance (in LD or FBD), RIGHT-click
   // to bring up the context menu and select "Open Instruction Logic".
   // This rung will appear with the STRING values for the selected instance.
   // You may double-click the STRING values here to modify them as well.
   // #####  V4.00.00  2018-07-16:  Added string for Cfg_Area, renamed Inf_* to HMI_*.  #####
   0: JMP(SkipText)LOWER(Cfg_Desc,Cfg_Label)LOWER(Cfg_Tag,Cfg_Area)LOWER(HMI_Lib,HMI_Type);
   // This rung handles received Command Source selection Inputs and Commands:
   // NOTE:  All Commands for Command Source and Alarm are aliased directly to the
   // corresponding Commands in the contained P_CmdSrc and P_Alarm AOIs.
   // #####  V4.00.00  2018-07-16:  Changed P_Mode to P_CmdSrc.  #####
   1: LBL(SkipText)P_CmdSrc(CmdSrc);
   // This rung handles simple First-Come First-Served Ownership Arbitration.
   // If a requestor supplies a non-zero Owner ID and the current owner is NONE (zero),
   // Ownership is assigned to the requesting ID.  When that requestor sets the Owner ID back
   // to zero, Ownership is relinquished back to NONE.
   2: [EQU(PSet_Owner,0) ,EQU(Val_Owner,0) ]MOV(PSet_Owner,Val_Owner);
   // ============================================================
   // CONFIGURATION
   // ============================================================
   // If the Valve does not have an Open Limit Switch input,
   // it cannot be used for Valve feedback checking.
   3: XIO(Cfg_HasOpenLS)OTU(Cfg_UseOpenLS);
   // If the Valve does not have a Closed Limit Switch input,
   // it cannot be used for Valve feedback checking.
   4: XIO(Cfg_HasClosedLS)OTU(Cfg_UseClosedLS);
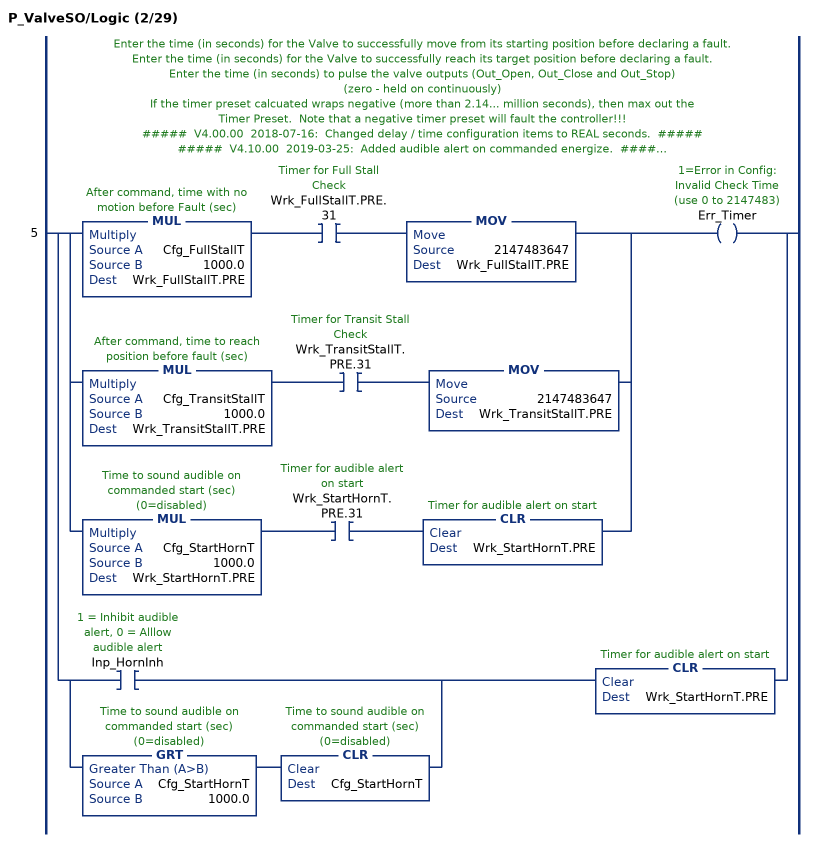
   // Enter the time (in seconds) for the Valve to successfully move from its starting position before declaring a fault.
   // Enter the time (in seconds) for the Valve to successfully reach its target position before declaring a fault.
   // Enter the time (in seconds) to pulse the valve outputs (Out_Open, Out_Close and Out_Stop)
   // (zero - held on continuously)
   // If the timer preset calcuated wraps negative (more than 2.14... million seconds), then max out the
   // Timer Preset.  Note that a negative timer preset will fault the controller!!!
   // #####  V4.00.00  2018-07-16:  Changed delay / time configuration items to REAL seconds.  #####
   // #####  V4.10.00  2019-03-25:  Added audible alert on commanded energize.  #####
   // #####  Added Inp_HornInh to disable Horn operation.  #####
   5: [[MUL(Cfg_FullStallT,1000.0,Wrk_FullStallT.PRE) XIC(Wrk_FullStallT.PRE.31) MOV(2147483647,Wrk_FullStallT.PRE) ,MUL(Cfg_TransitStallT,1000.0,Wrk_TransitStallT.PRE) XIC(Wrk_TransitStallT.PRE.31) MOV(2147483647,Wrk_TransitStallT.PRE) ,MUL(Cfg_StartHornT,1000.0,Wrk_StartHornT.PRE) XIC(Wrk_StartHornT.PRE.31) CLR(Wrk_StartHornT.PRE) ] OTE(Err_Timer) ,[XIC(Inp_HornInh) ,GRT(Cfg_StartHornT,1000.0) CLR(Cfg_StartHornT) ] CLR(Wrk_StartHornT.PRE) ];
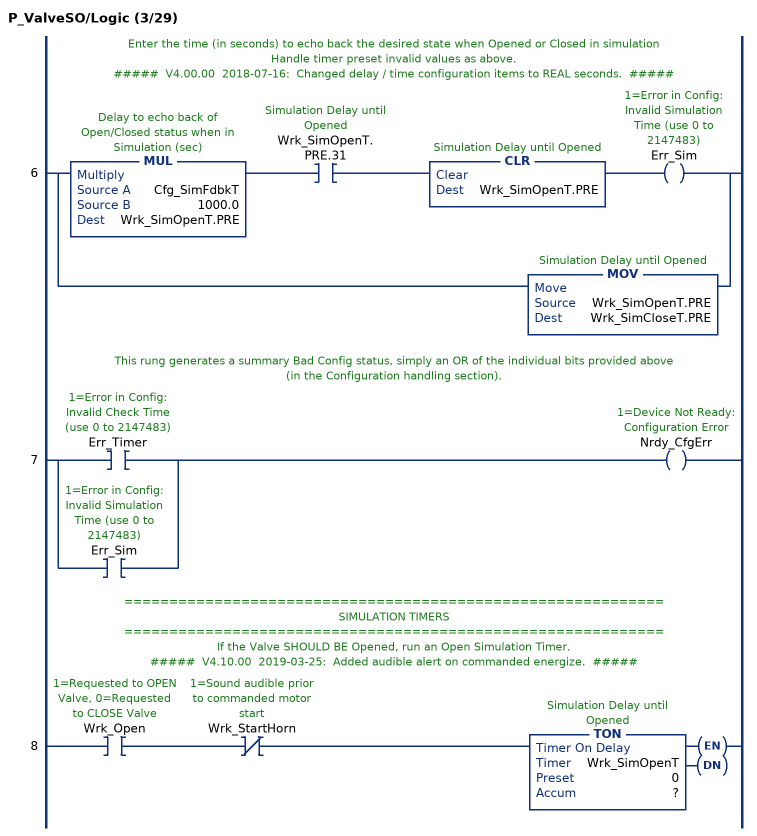
   // Enter the time (in seconds) to echo back the desired state when Opened or Closed in simulation
   // Handle timer preset invalid values as above.
   // #####  V4.00.00  2018-07-16:  Changed delay / time configuration items to REAL seconds.  #####
   6: [MUL(Cfg_SimFdbkT,1000.0,Wrk_SimOpenT.PRE) XIC(Wrk_SimOpenT.PRE.31) CLR(Wrk_SimOpenT.PRE) OTE(Err_Sim) ,MOV(Wrk_SimOpenT.PRE,Wrk_SimCloseT.PRE) ];
   // This rung generates a summary Bad Config status, simply an OR of the individual bits provided above
   // (in the Configuration handling section).
   7: [XIC(Err_Timer) ,XIC(Err_Sim) ]OTE(Nrdy_CfgErr);
   // ============================================================
   // SIMULATION TIMERS
   // ============================================================
   // If the Valve SHOULD BE Opened, run an Open Simulation Timer.
   // #####  V4.10.00  2019-03-25:  Added audible alert on commanded energize.  #####
   8: XIC(Wrk_Open)XIO(Wrk_StartHorn)TON(Wrk_SimOpenT,?,?);
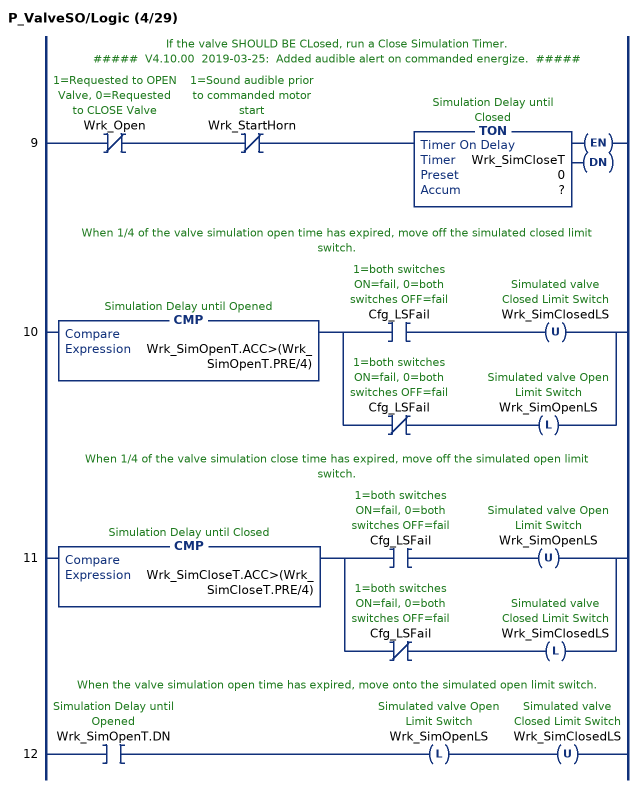
   // If the valve SHOULD BE CLosed, run a Close Simulation Timer.
   // #####  V4.10.00  2019-03-25:  Added audible alert on commanded energize.  #####
   9: XIO(Wrk_Open)XIO(Wrk_StartHorn)TON(Wrk_SimCloseT,?,?);
   // When 1/4 of the valve simulation open time has expired, move off the simulated closed limit switch.
   10: CMP(Wrk_SimOpenT.ACC>(Wrk_SimOpenT.PRE/4))[XIC(Cfg_LSFail) OTU(Wrk_SimClosedLS) ,XIO(Cfg_LSFail) OTL(Wrk_SimOpenLS) ];
   // When 1/4 of the valve simulation close time has expired, move off the simulated open limit switch.
   11: CMP(Wrk_SimCloseT.ACC>(Wrk_SimCloseT.PRE/4))[XIC(Cfg_LSFail) OTU(Wrk_SimOpenLS) ,XIO(Cfg_LSFail) OTL(Wrk_SimClosedLS) ];
   // When the valve simulation open time has expired, move onto the simulated open limit switch.
   12: XIC(Wrk_SimOpenT.DN)OTL(Wrk_SimOpenLS)OTU(Wrk_SimClosedLS);
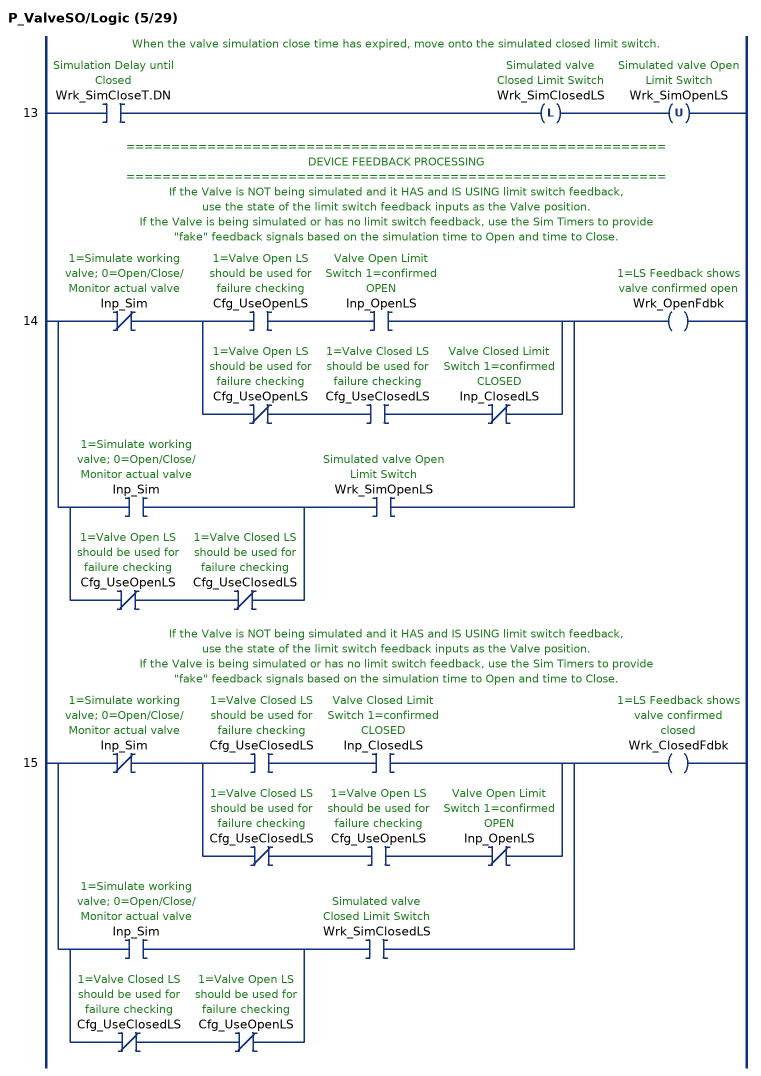
   // When the valve simulation close time has expired, move onto the simulated closed limit switch.
   13: XIC(Wrk_SimCloseT.DN)OTL(Wrk_SimClosedLS)OTU(Wrk_SimOpenLS);
   // ============================================================
   // DEVICE FEEDBACK PROCESSING
   // ============================================================
   // If the Valve is NOT being simulated and it HAS and IS USING limit switch feedback,
   // use the state of the limit switch feedback inputs as the Valve position.
   // If the Valve is being simulated or has no limit switch feedback, use the Sim Timers to provide
   // "fake" feedback signals based on the simulation time to Open and time to Close.
   14: [XIO(Inp_Sim) [XIC(Cfg_UseOpenLS) XIC(Inp_OpenLS) ,XIO(Cfg_UseOpenLS) XIC(Cfg_UseClosedLS) XIO(Inp_ClosedLS) ] ,[XIC(Inp_Sim) ,XIO(Cfg_UseOpenLS) XIO(Cfg_UseClosedLS) ] XIC(Wrk_SimOpenLS) ]OTE(Wrk_OpenFdbk);
   // If the Valve is NOT being simulated and it HAS and IS USING limit switch feedback,
   // use the state of the limit switch feedback inputs as the Valve position.
   // If the Valve is being simulated or has no limit switch feedback, use the Sim Timers to provide
   // "fake" feedback signals based on the simulation time to Open and time to Close.
   15: [XIO(Inp_Sim) [XIC(Cfg_UseClosedLS) XIC(Inp_ClosedLS) ,XIO(Cfg_UseClosedLS) XIC(Cfg_UseOpenLS) XIO(Inp_OpenLS) ] ,[XIC(Inp_Sim) ,XIO(Cfg_UseClosedLS) XIO(Cfg_UseOpenLS) ] XIC(Wrk_SimClosedLS) ]OTE(Wrk_ClosedFdbk);
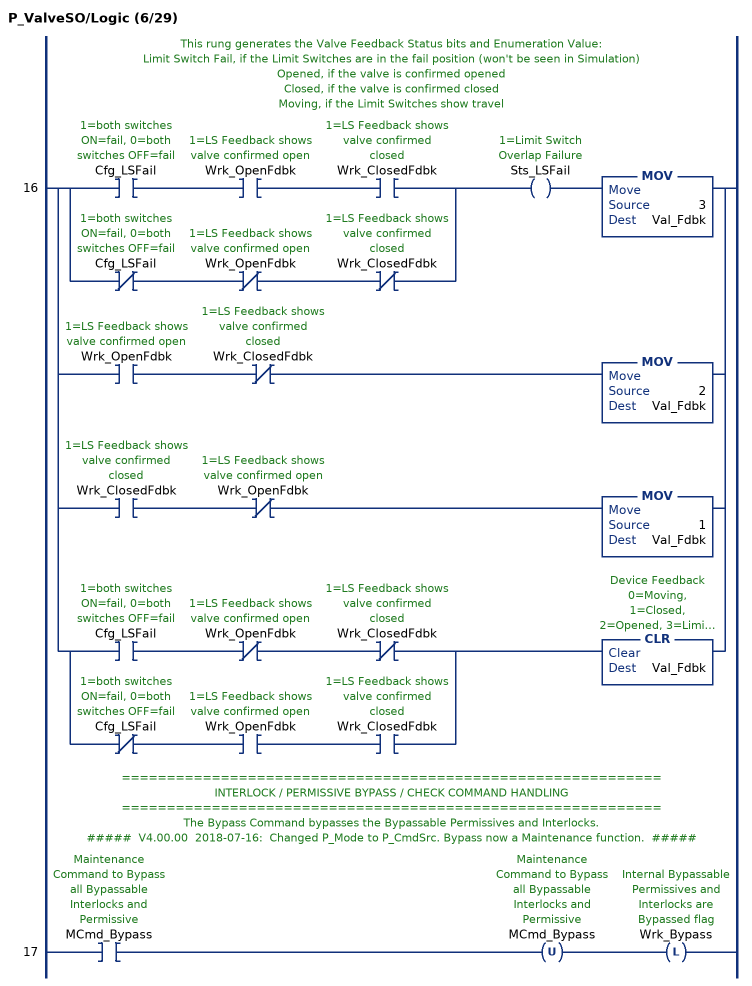
   // This rung generates the Valve Feedback Status bits and Enumeration Value:
   // Limit Switch Fail, if the Limit Switches are in the fail position (won't be seen in Simulation)
   // Opened, if the valve is confirmed opened
   // Closed, if the valve is confirmed closed
   // Moving, if the Limit Switches show travel
   16: [[XIC(Cfg_LSFail) XIC(Wrk_OpenFdbk) XIC(Wrk_ClosedFdbk) ,XIO(Cfg_LSFail) XIO(Wrk_OpenFdbk) XIO(Wrk_ClosedFdbk) ] OTE(Sts_LSFail) MOV(3,Val_Fdbk) ,XIC(Wrk_OpenFdbk) XIO(Wrk_ClosedFdbk) MOV(2,Val_Fdbk) ,XIC(Wrk_ClosedFdbk) XIO(Wrk_OpenFdbk) MOV(1,Val_Fdbk) ,[XIC(Cfg_LSFail) XIO(Wrk_OpenFdbk) XIO(Wrk_ClosedFdbk) ,XIO(Cfg_LSFail) XIC(Wrk_OpenFdbk) XIC(Wrk_ClosedFdbk) ] CLR(Val_Fdbk) ];
   // ============================================================
   // INTERLOCK / PERMISSIVE BYPASS / CHECK COMMAND HANDLING
   // ============================================================
   // The Bypass Command bypasses the Bypassable Permissives and Interlocks.
   // #####  V4.00.00  2018-07-16:  Changed P_Mode to P_CmdSrc. Bypass now a Maintenance function.  #####
   17: XIC(MCmd_Bypass)OTU(MCmd_Bypass)OTL(Wrk_Bypass);
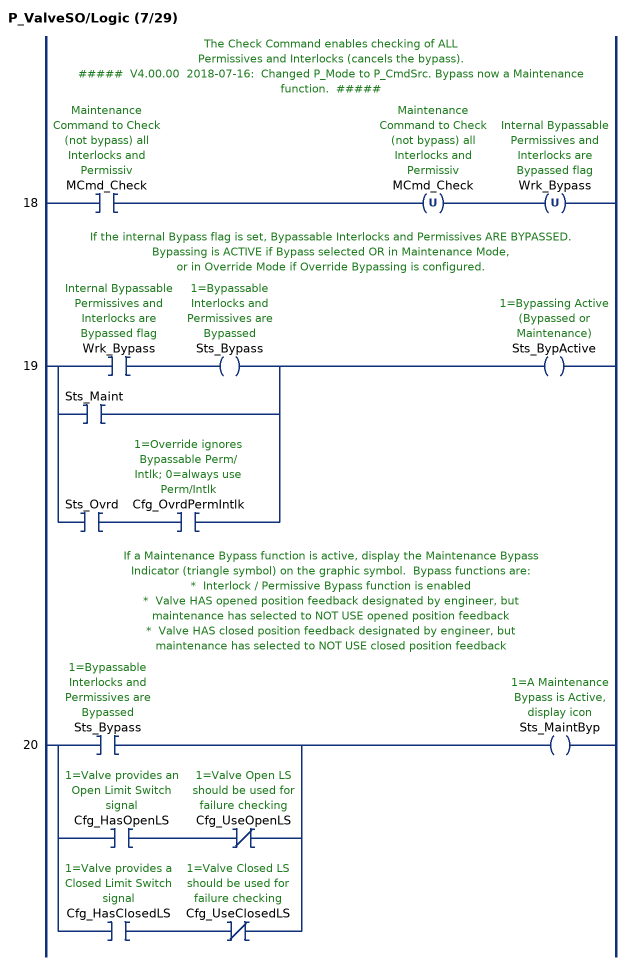
   // The Check Command enables checking of ALL
   // Permissives and Interlocks (cancels the bypass).
   // #####  V4.00.00  2018-07-16:  Changed P_Mode to P_CmdSrc. Bypass now a Maintenance function.  #####
   18: XIC(MCmd_Check)OTU(MCmd_Check)OTU(Wrk_Bypass);
   // If the internal Bypass flag is set, Bypassable Interlocks and Permissives ARE BYPASSED.
   // Bypassing is ACTIVE if Bypass selected OR in Maintenance Mode,
   // or in Override Mode if Override Bypassing is configured.
   19: [XIC(Wrk_Bypass) OTE(Sts_Bypass) ,XIC(Sts_Maint) ,XIC(Sts_Ovrd) XIC(Cfg_OvrdPermIntlk) ]OTE(Sts_BypActive);
   // If a Maintenance Bypass function is active, display the Maintenance Bypass
   // Indicator (triangle symbol) on the graphic symbol.  Bypass functions are:
   // *  Interlock / Permissive Bypass function is enabled
   // *  Valve HAS opened position feedback designated by engineer, but
   // maintenance has selected to NOT USE opened position feedback
   // *  Valve HAS closed position feedback designated by engineer, but
   // maintenance has selected to NOT USE closed position feedback
   20: [XIC(Sts_Bypass) ,XIC(Cfg_HasOpenLS) XIO(Cfg_UseOpenLS) ,XIC(Cfg_HasClosedLS) XIO(Cfg_UseClosedLS) ]OTE(Sts_MaintByp);
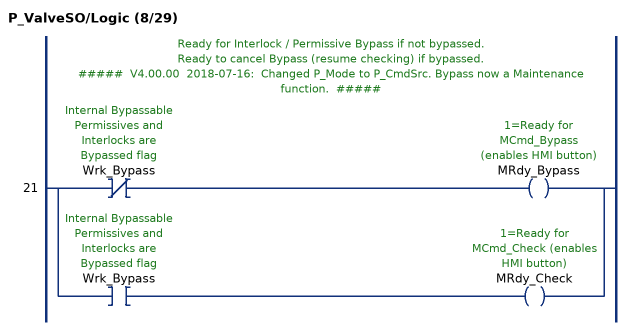
   // Ready for Interlock / Permissive Bypass if not bypassed.
   // Ready to cancel Bypass (resume checking) if bypassed.
   // #####  V4.00.00  2018-07-16:  Changed P_Mode to P_CmdSrc. Bypass now a Maintenance function.  #####
   21: [XIO(Wrk_Bypass) OTE(MRdy_Bypass) ,XIC(Wrk_Bypass) OTE(MRdy_Check) ];
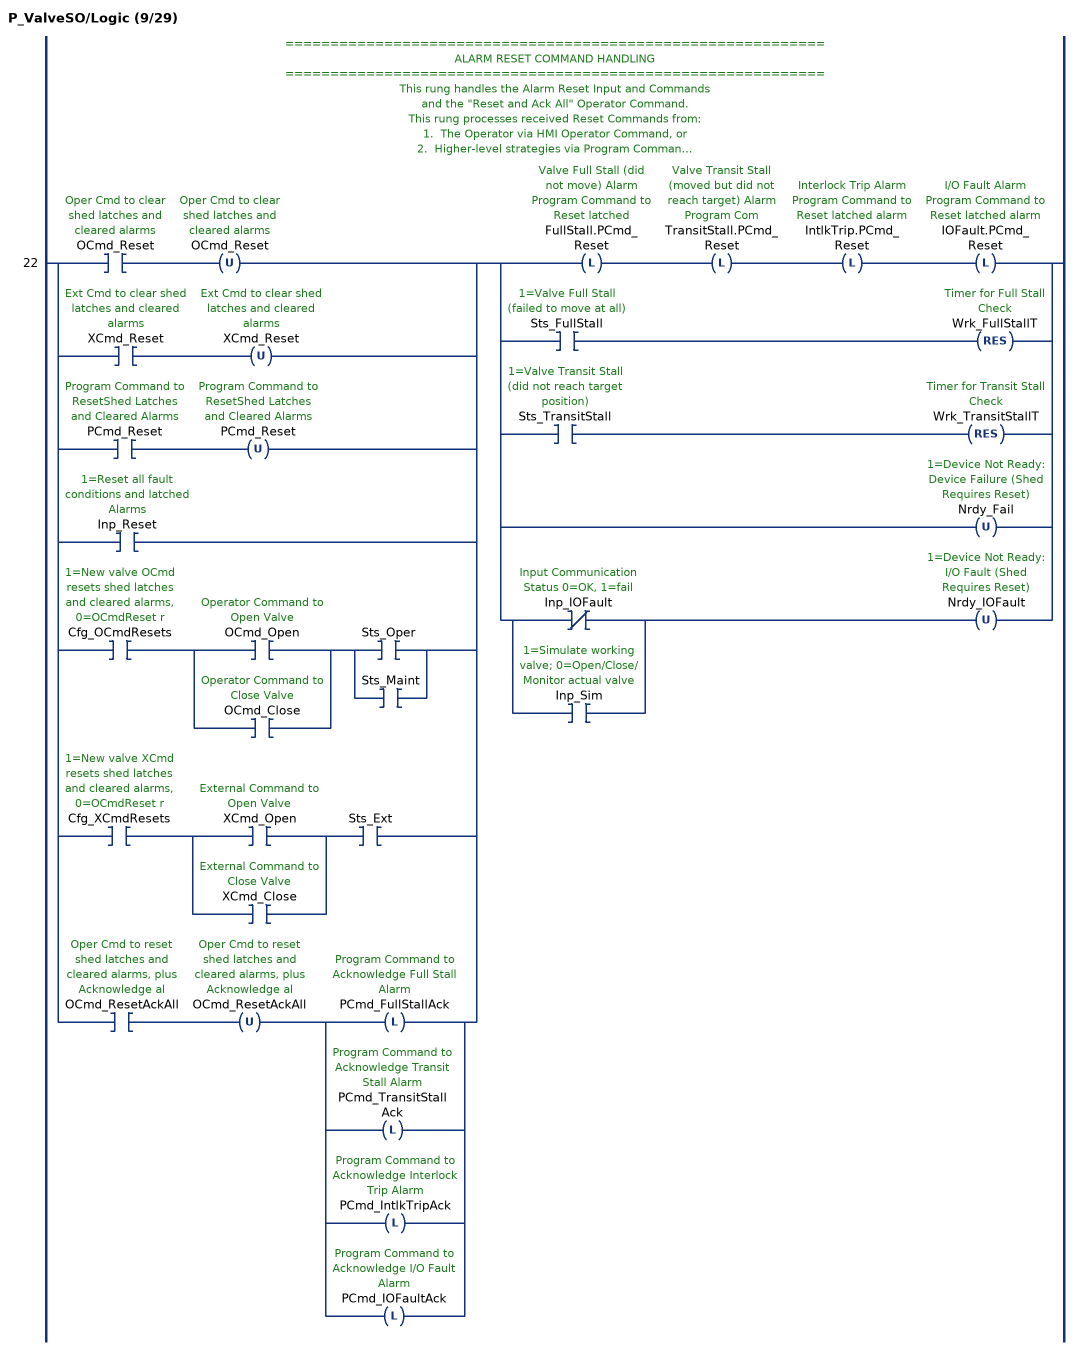
   // ============================================================
   // ALARM RESET COMMAND HANDLING
   // ============================================================
   // This rung handles the Alarm Reset Input and Commands
   // and the "Reset and Ack All" Operator Command.
   // This rung processes received Reset Commands from:
   // 1.  The Operator via HMI Operator Command, or
   // 2.  Higher-level strategies via Program Command
   // 3.  Pushbuttons or other block via Input
   // 4.  Resets initiated by other device Operator Commands (if configured to do so)
   // and forwards the Reset to ALL Alarms and latched Shed conditions.
   // #####  V4.00.00  2018-07-16:  Deleted Cfg_PCmdClear; all Program Commands are now self-clearing.  #####
   // #####  Added External Command Source and Commands.  #####
   // #####  V4.00.01  2018-08-24:  Corrected Reset Command logic.  #####
   22: [XIC(OCmd_Reset) OTU(OCmd_Reset) ,XIC(XCmd_Reset) OTU(XCmd_Reset) ,XIC(PCmd_Reset) OTU(PCmd_Reset) ,XIC(Inp_Reset) ,XIC(Cfg_OCmdResets) [XIC(OCmd_Open) ,XIC(OCmd_Close) ] [XIC(Sts_Oper) ,XIC(Sts_Maint) ] ,XIC(Cfg_XCmdResets) [XIC(XCmd_Open) ,XIC(XCmd_Close) ] XIC(Sts_Ext) ,XIC(OCmd_ResetAckAll) OTU(OCmd_ResetAckAll) [OTL(PCmd_FullStallAck) ,OTL(PCmd_TransitStallAck) ,OTL(PCmd_IntlkTripAck) ,OTL(PCmd_IOFaultAck) ] ][OTL(FullStall.PCmd_Reset) OTL(TransitStall.PCmd_Reset) OTL(IntlkTrip.PCmd_Reset) OTL(IOFault.PCmd_Reset) ,XIC(Sts_FullStall) RES(Wrk_FullStallT) ,XIC(Sts_TransitStall) RES(Wrk_TransitStallT) ,OTU(Nrdy_Fail) ,[XIO(Inp_IOFault) ,XIC(Inp_Sim) ] OTU(Nrdy_IOFault) ];
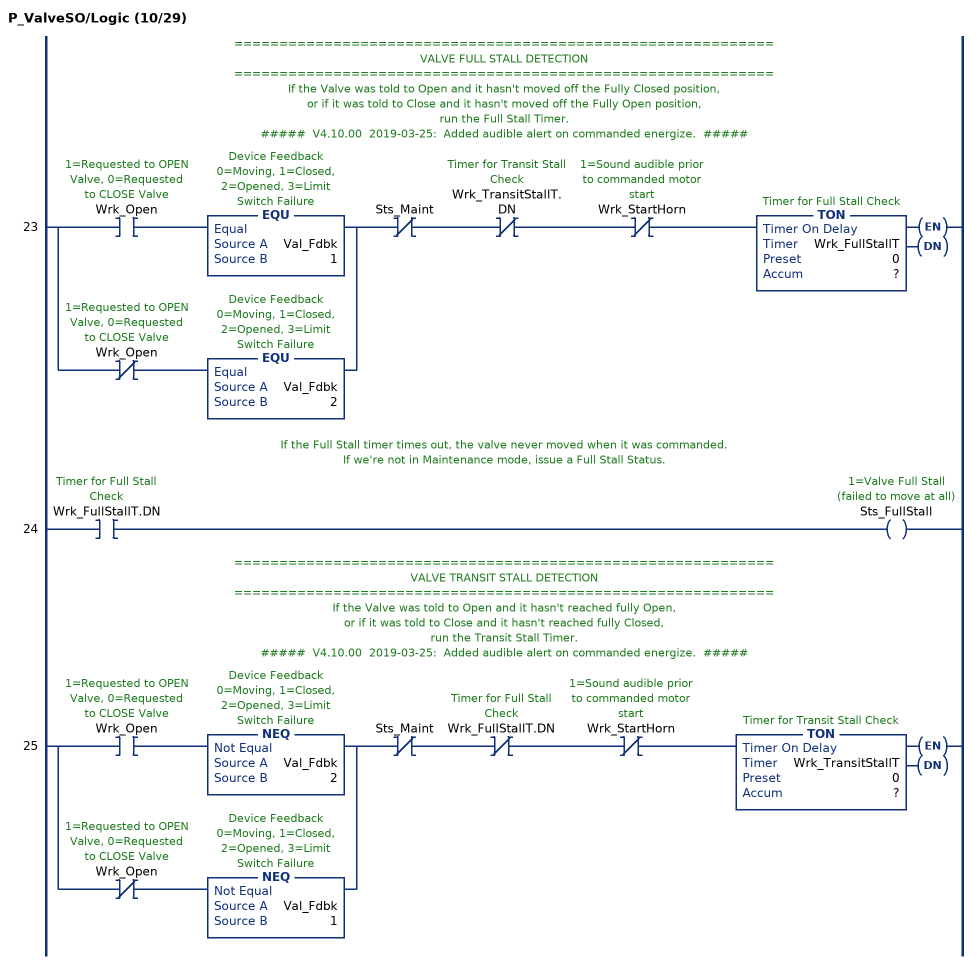
   // ============================================================
   // VALVE FULL STALL DETECTION
   // ============================================================
   // If the Valve was told to Open and it hasn't moved off the Fully Closed position,
   // or if it was told to Close and it hasn't moved off the Fully Open position,
   // run the Full Stall Timer.
   // #####  V4.10.00  2019-03-25:  Added audible alert on commanded energize.  #####
   23: [XIC(Wrk_Open) EQU(Val_Fdbk,1) ,XIO(Wrk_Open) EQU(Val_Fdbk,2) ]XIO(Sts_Maint)XIO(Wrk_TransitStallT.DN)XIO(Wrk_StartHorn)TON(Wrk_FullStallT,?,?);
   // If the Full Stall timer times out, the valve never moved when it was commanded.
   // If we're not in Maintenance mode, issue a Full Stall Status.
   24: XIC(Wrk_FullStallT.DN)OTE(Sts_FullStall);
   // ============================================================
   // VALVE TRANSIT STALL DETECTION
   // ============================================================
   // If the Valve was told to Open and it hasn't reached fully Open,
   // or if it was told to Close and it hasn't reached fully Closed,
   // run the Transit Stall Timer.
   // #####  V4.10.00  2019-03-25:  Added audible alert on commanded energize.  #####
   25: [XIC(Wrk_Open) NEQ(Val_Fdbk,2) ,XIO(Wrk_Open) NEQ(Val_Fdbk,1) ]XIO(Sts_Maint)XIO(Wrk_FullStallT.DN)XIO(Wrk_StartHorn)TON(Wrk_TransitStallT,?,?);
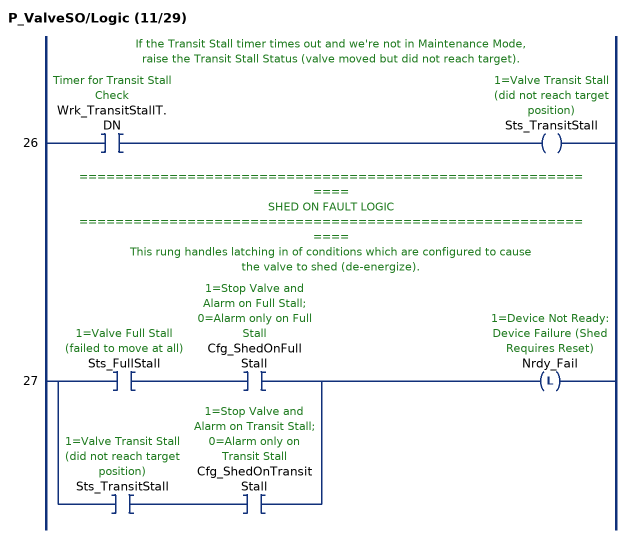
   // If the Transit Stall timer times out and we're not in Maintenance Mode,
   // raise the Transit Stall Status (valve moved but did not reach target).
   26: XIC(Wrk_TransitStallT.DN)OTE(Sts_TransitStall);
   // ============================================================
   // SHED ON FAULT LOGIC
   // ============================================================
   // This rung handles latching in of conditions which are configured to cause
   // the valve to shed (de-energize).
   27: [XIC(Sts_FullStall) XIC(Cfg_ShedOnFullStall) ,XIC(Sts_TransitStall) XIC(Cfg_ShedOnTransitStall) ]OTL(Nrdy_Fail);
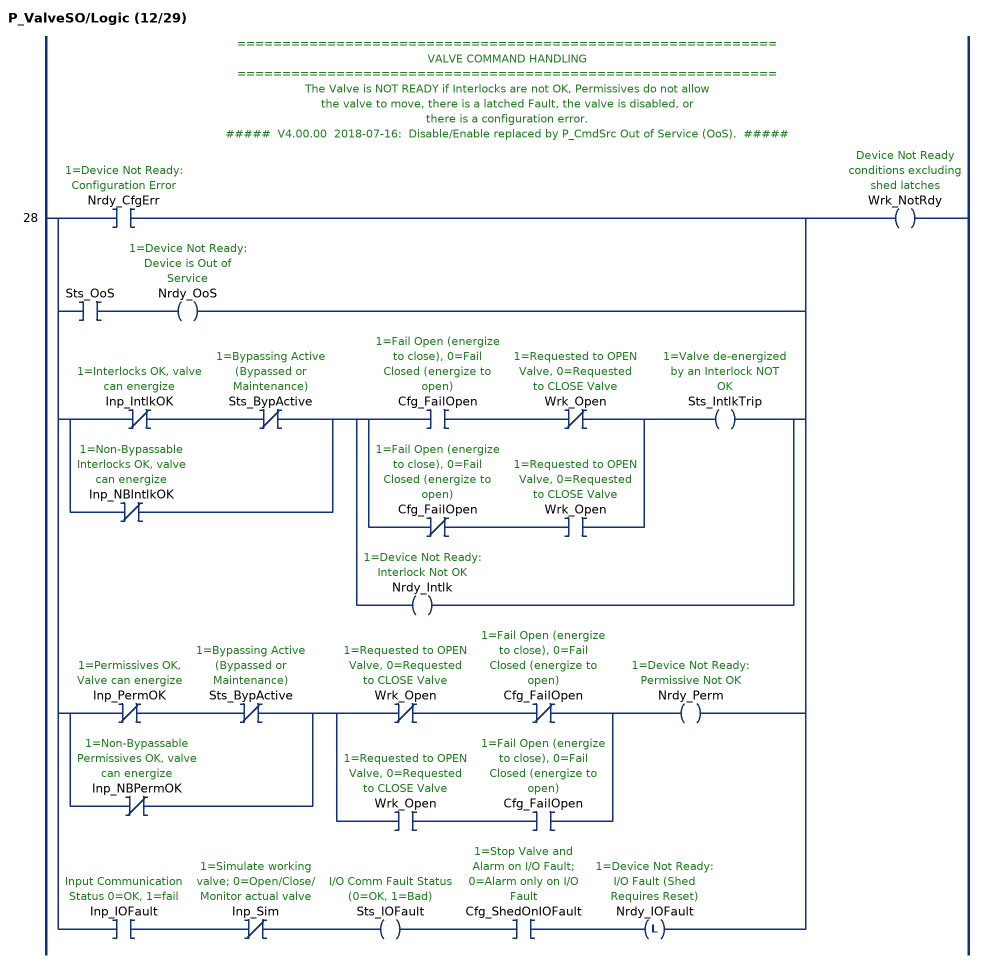
   // ============================================================
   // VALVE COMMAND HANDLING
   // ============================================================
   // The Valve is NOT READY if Interlocks are not OK, Permissives do not allow
   // the valve to move, there is a latched Fault, the valve is disabled, or
   // there is a configuration error.
   // #####  V4.00.00  2018-07-16:  Disable/Enable replaced by P_CmdSrc Out of Service (OoS).  #####
   28: [XIC(Nrdy_CfgErr) ,XIC(Sts_OoS) OTE(Nrdy_OoS) ,[XIO(Inp_IntlkOK) XIO(Sts_BypActive) ,XIO(Inp_NBIntlkOK) ] [[XIC(Cfg_FailOpen) XIO(Wrk_Open) ,XIO(Cfg_FailOpen) XIC(Wrk_Open) ] OTE(Sts_IntlkTrip) ,OTE(Nrdy_Intlk) ] ,[XIO(Inp_PermOK) XIO(Sts_BypActive) ,XIO(Inp_NBPermOK) ] [XIO(Wrk_Open) XIO(Cfg_FailOpen) ,XIC(Wrk_Open) XIC(Cfg_FailOpen) ] OTE(Nrdy_Perm) ,XIC(Inp_IOFault) XIO(Inp_Sim) OTE(Sts_IOFault) XIC(Cfg_ShedOnIOFault) OTL(Nrdy_IOFault) ]OTE(Wrk_NotRdy);
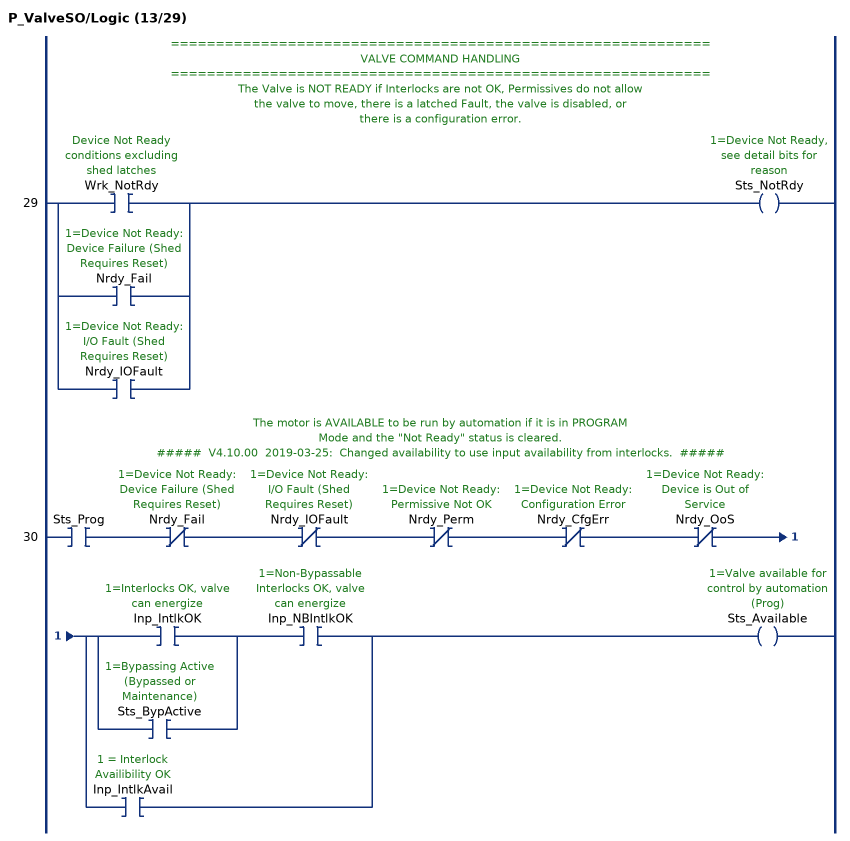
   // ============================================================
   // VALVE COMMAND HANDLING
   // ============================================================
   // The Valve is NOT READY if Interlocks are not OK, Permissives do not allow
   // the valve to move, there is a latched Fault, the valve is disabled, or
   // there is a configuration error.
   29: [XIC(Wrk_NotRdy) ,XIC(Nrdy_Fail) ,XIC(Nrdy_IOFault) ]OTE(Sts_NotRdy);
   // The motor is AVAILABLE to be run by automation if it is in PROGRAM
   // Mode and the "Not Ready" status is cleared.
   // #####  V4.10.00  2019-03-25:  Changed availability to use input availability from interlocks.  #####
   30: XIC(Sts_Prog)XIO(Nrdy_Fail)XIO(Nrdy_IOFault)XIO(Nrdy_Perm)XIO(Nrdy_CfgErr)XIO(Nrdy_OoS)[[XIC(Inp_IntlkOK) ,XIC(Sts_BypActive) ] XIC(Inp_NBIntlkOK) ,XIC(Inp_IntlkAvail) ]OTE(Sts_Available);
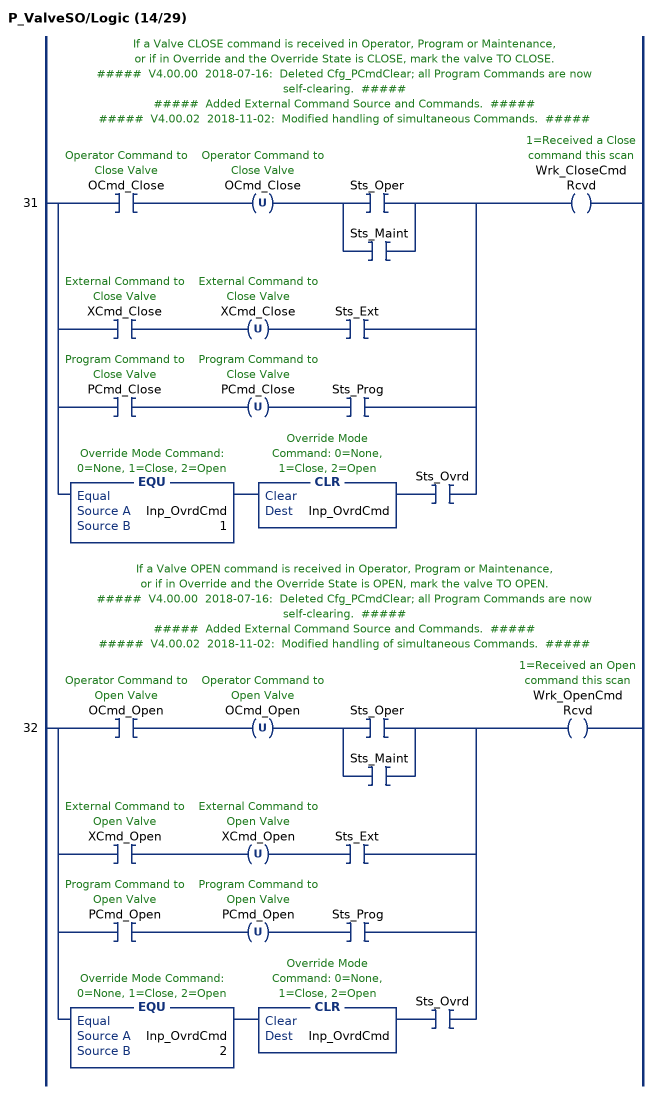
   // If a Valve CLOSE command is received in Operator, Program or Maintenance,
   // or if in Override and the Override State is CLOSE, mark the valve TO CLOSE.
   // #####  V4.00.00  2018-07-16:  Deleted Cfg_PCmdClear; all Program Commands are now self-clearing.  #####
   // #####  Added External Command Source and Commands.  #####
   // #####  V4.00.02  2018-11-02:  Modified handling of simultaneous Commands.  #####
   31: [XIC(OCmd_Close) OTU(OCmd_Close) [XIC(Sts_Oper) ,XIC(Sts_Maint) ] ,XIC(XCmd_Close) OTU(XCmd_Close) XIC(Sts_Ext) ,XIC(PCmd_Close) OTU(PCmd_Close) XIC(Sts_Prog) ,EQU(Inp_OvrdCmd,1) CLR(Inp_OvrdCmd) XIC(Sts_Ovrd) ]OTE(Wrk_CloseCmdRcvd);
   // If a Valve OPEN command is received in Operator, Program or Maintenance,
   // or if in Override and the Override State is OPEN, mark the valve TO OPEN.
   // #####  V4.00.00  2018-07-16:  Deleted Cfg_PCmdClear; all Program Commands are now self-clearing.  #####
   // #####  Added External Command Source and Commands.  #####
   // #####  V4.00.02  2018-11-02:  Modified handling of simultaneous Commands.  #####
   32: [XIC(OCmd_Open) OTU(OCmd_Open) [XIC(Sts_Oper) ,XIC(Sts_Maint) ] ,XIC(XCmd_Open) OTU(XCmd_Open) XIC(Sts_Ext) ,XIC(PCmd_Open) OTU(PCmd_Open) XIC(Sts_Prog) ,EQU(Inp_OvrdCmd,2) CLR(Inp_OvrdCmd) XIC(Sts_Ovrd) ]OTE(Wrk_OpenCmdRcvd);
